LIN {X 0,Y 530.986,Z 634.341,A -85,B 0,C 180,E1 -4457.833,E2 -4457.833} C_VEL
LIN {X 0,Y 531.019,Z 634.341,A -85,B 0,C 180,E1 -4460.559,E2 -4460.559} C_VEL
LIN {X 0,Y 530.968,Z 634.345,A -85,B 0,C 180,E1 -4463.842,E2 -4463.842} C_VEL
LIN {X 0,Y 530.995,Z 634.341,A -85,B 0,C 180,E1 -4466.494,E2 -4466.494} C_VEL
LIN {X 0,Y 530.979,Z 634.341,A -85,B 0,C 180,E1 -4469.353,E2 -4469.353} C_VEL
LIN {X 0,Y 531.014,Z 634.337,A -85,B 0,C 180,E1 -4472.404,E2 -4472.404} C_VEL
LIN {X 0,Y 531.004,Z 634.337,A -85,B 0,C 180,E1 -4474.942,E2 -4474.942} C_VEL
LIN {X 0,Y 530.967,Z 634.342,A -85,B 0,C 180,E1 -4478.246,E2 -4478.246} C_VEL
LIN {X 0,Y 530.993,Z 634.339,A -85,B 0,C 180,E1 -4480.677,E2 -4480.677} C_VEL
LIN {X 0,Y 530.982,Z 634.346,A -85,B 0,C 180,E1 -4483.071,E2 -4483.071} C_VEL
LIN {X 0,Y 531.014,Z 634.339,A -85,B 0,C 180,E1 -4485.436,E2 -4485.436} C_VEL
LIN {X 0,Y 531.042,Z 634.337,A -85,B 0,C 180,E1 -4488.55,E2 -4488.55} C_VEL
LIN {X 0,Y 531.056,Z 634.331,A -85,B 0,C 180,E1 -4491.629,E2 -4491.629} C_VEL
LIN {X 0,Y 531.118,Z 634.33,A -85,B 0,C 180,E1 -4494.685,E2 -4494.685} C_VEL
LIN {X 0,Y 531.134,Z 634.323,A -85,B 0,C 180,E1 -4497.725,E2 -4497.725} C_VEL
LIN {X 0,Y 531.149,Z 634.323,A -85,B 0,C 180,E1 -4500.758,E2 -4500.758} C_VEL
LIN {X 0,Y 531.105,Z 634.328,A -85,B 0,C 180,E1 -4503.034,E2 -4503.034} C_VEL
LIN {X 0,Y 531.06,Z 634.46,A -85,B 0,C 180,E1 -4504.649,E2 -4504.649} C_VEL
LIN {X 0,Y 531.55,Z 640.442,A -85,B 0,C 180,E1 -4506.072,E2 -4506.072} C_VEL
LIN {X 0,Y 531.68,Z 653.246,A -85,B 0,C 180,E1 -4509.127,E2 -4509.127} C_VEL
LIN {X 0,Y 531.676,Z 665.851,A -85,B 0,C 180,E1 -4512.21,E2 -4512.21} C_VEL
LIN {X 0,Y 531.52,Z 677.588,A -85,B 0,C 180,E1 -4515.154,E2 -4515.154} C_VEL
LIN {X 0,Y 531.397,Z 689.132,A -85,B 0,C 180,E1 -4518.067,E2 -4518.067} C_VEL
LIN {X 0,Y 531.209,Z 700.198,A -85,B 0,C 180,E1 -4520.929,E2 -4520.929} C_VEL
LIN {X 0,Y 531.024,Z 710.926,A -85,B 0,C 180,E1 -4523.717,E2 -4523.717} C_VEL
LIN {X 0,Y 530.877,Z 722.756,A -85,B 0,C 180,E1 -4526.751,E2 -4526.751} C_VEL
LIN {X 0,Y 530.807,Z 725.673,A -85,B 0,C 180,E1 -4527.491,E2 -4527.491} C_VEL
LIN {X 0,Y 532.339,Z 736.306,A -85,B 0,C 180,E1 -4527.756,E2 -4527.756} C_VEL
LIN {X 0,Y 532.152,Z 749.102,A -85,B 0,C 180,E1 -4528.152,E2 -4528.152} C_VEL
LIN {X 0,Y 531.867,Z 762.095,A -85,B 0,C 180,E1 -4528.728,E2 -4528.728} C_VEL
LIN {X 0,Y 531.627,Z 773.458,A -85,B 0,C 180,E1 -4529.392,E2 -4529.392} C_VEL
LIN {X 0,Y 531.387,Z 783.981,A -85,B 0,C 180,E1 -4530.171,E2 -4530.171} C_VEL
LIN {X 0,Y 531.104,Z 794.919,A -85,B 0,C 180,E1 -4531.18,E2 -4531.18} C_VEL
LIN {X 0,Y 530.918,Z 804.119,A -85,B 0,C 180,E1 -4532.24,E2 -4532.24} C_VEL
LIN {X 0,Y 530.742,Z 812.635,A -85,B 0,C 180,E1 -4533.465,E2 -4533.465} C_VEL
LIN {X 0,Y 530.587,Z 819.541,A -85,B 0,C 180,E1 -4534.72,E2 -4534.72} C_VEL
LIN {X 0,Y 530.57,Z 820.437,A -85,B 0,C 180,E1 -4534.911,E2 -4534.911} C_VEL
LIN {X 0,Y 529.876,Z 823.006,A -85,B 0,C 180,E1 -4535.484,E2 -4535.484} C_VEL
LIN {X 0,Y 526.94,Z 826.619,A -85,B 0,C 180,E1 -4536.435,E2 -4536.435} C_VEL
LIN {X 0,Y 524.46,Z 828.999,A -85,B 0,C 180,E1 -4537.22,E2 -4537.22} C_VEL
LIN {X 0,Y 523.384,Z 830.509,A -85,B 0,C 180,E1 -4537.836,E2 -4537.836} C_VEL
LIN {X 0,Y 523.29,Z 830.939,A -85,B 0,C 180,E1 -4538.047,E2 -4538.047} C_VEL
LIN {X 0,Y 523.257,Z 832.782,A -85,B 0,C 180,E1 -4539.144,E2 -4539.144} C_VEL
LIN {X 0,Y 523.237,Z 833.705,A -85,B 0,C 180,E1 -4540.145,E2 -4540.145} C_VEL
LIN {X 0,Y 523.242,Z 833.97,A -85,B 0,C 180,E1 -4541.222,E2 -4541.222} C_VEL
LIN {X 0,Y 523.262,Z 833.392,A -85,B 0,C 180,E1 -4542.379,E2 -4542.379} C_VEL
LIN {X 0,Y 523.26,Z 831.963,A -85,B 0,C 180,E1 -4543.509,E2 -4543.509} C_VEL
LIN {X 0,Y 523.362,Z 828.741,A -85,B 0,C 180,E1 -4544.974,E2 -4544.974} C_VEL
LIN {X 0,Y 523.418,Z 825.122,A -85,B 0,C 180,E1 -4546.12,E2 -4546.12} C_VEL
LIN {X 0,Y 523.493,Z 820.639,A -85,B 0,C 180,E1 -4547.218,E2 -4547.218} C_VEL
LIN {X 0,Y 523.636,Z 813.716,A -85,B 0,C 180,E1 -4548.551,E2 -4548.551} C_VEL
LIN {X 0,Y 523.816,Z 806.45,A -85,B 0,C 180,E1 -4549.658,E2 -4549.658} C_VEL
LIN {X 0,Y 524.007,Z 797.164,A -85,B 0,C 180,E1 -4550.8,E2 -4550.8} C_VEL
LIN {X 0,Y 524.268,Z 787.013,A -85,B 0,C 180,E1 -4551.807,E2 -4551.807} C_VEL
LIN {X 0,Y 524.587,Z 775.831,A -85,B 0,C 180,E1 -4552.69,E2 -4552.69} C_VEL
LIN {X 0,Y 524.854,Z 764.914,A -85,B 0,C 180,E1 -4553.376,E2 -4553.376} C_VEL
LIN {X 0,Y 525.154,Z 753.694,A -85,B 0,C 180,E1 -4553.926,E2 -4553.926} C_VEL
LIN {X 0,Y 525.392,Z 740.78,A -85,B 0,C 180,E1 -4554.388,E2 -4554.388} C_VEL
LIN {X 0,Y 525.236,Z 734.832,A -85,B 0,C 180,E1 -4554.553,E2 -4554.553} C_VEL
LIN {X 0,Y 523.71,Z 725.662,A -85,B 0,C 180,E1 -4554.789,E2 -4554.789} C_VEL
LIN {X 0,Y 523.937,Z 714.498,A -85,B 0,C 180,E1 -4557.679,E2 -4557.679} C_VEL
LIN {X 0,Y 524.166,Z 703.144,A -85,B 0,C 180,E1 -4560.635,E2 -4560.635} C_VEL
LIN {X 0,Y 524.387,Z 690.741,A -85,B 0,C 180,E1 -4563.891,E2 -4563.891} C_VEL
LIN {X 0,Y 524.587,Z 679.935,A -85,B 0,C 180,E1 -4566.721,E2 -4566.721} C_VEL
LIN {X 0,Y 524.755,Z 668.733,A -85,B 0,C 180,E1 -4569.637,E2 -4569.637} C_VEL
LIN {X 0,Y 524.836,Z 657.835,A -85,B 0,C 180,E1 -4572.465,E2 -4572.465} C_VEL
LIN {X 0,Y 524.902,Z 647.071,A -85,B 0,C 180,E1 -4575.263,E2 -4575.263} C_VEL
LIN {X 0,Y 524.69,Z 639.508,A -85,B 0,C 180,E1 -4577.232,E2 -4577.232} C_VEL
LIN {X 0,Y 524.013,Z 635.215,A -85,B 0,C 180,E1 -4578.395,E2 -4578.395} C_VEL
LIN {X 0,Y 524.007,Z 635.217,A -85,B 0,C 180,E1 -4581.517,E2 -4581.517} C_VEL
LIN {X 0,Y 524.086,Z 635.205,A -85,B 0,C 180,E1 -4584.614,E2 -4584.614} C_VEL
LIN {X 0,Y 524.114,Z 635.202,A -85,B 0,C 180,E1 -4587.695,E2 -4587.695} C_VEL
LIN {X 0,Y 524.127,Z 635.201,A -85,B 0,C 180,E1 -4590.769,E2 -4590.769} C_VEL
LIN {X 0,Y 524.075,Z 635.206,A -85,B 0,C 180,E1 -4593.075,E2 -4593.075} C_VEL
LIN {X 0,Y 524.039,Z 635.21,A -85,B 0,C 180,E1 -4596.159,E2 -4596.159} C_VEL
LIN {X 0,Y 524.008,Z 635.215,A -85,B 0,C 180,E1 -4598.484,E2 -4598.484} C_VEL
LIN {X 0,Y 524.027,Z 635.211,A -85,B 0,C 180,E1 -4601.752,E2 -4601.752} C_VEL
LIN {X 0,Y 523.995,Z 635.216,A -85,B 0,C 180,E1 -4605.053,E2 -4605.053} C_VEL
LIN {X 0,Y 523.966,Z 635.222,A -85,B 0,C 180,E1 -4607.969,E2 -4607.969} C_VEL
LIN {X 0,Y 523.974,Z 635.22,A -85,B 0,C 180,E1 -4610.41,E2 -4610.41} C_VEL
LIN {X 0,Y 523.913,Z 635.226,A -85,B 0,C 180,E1 -4612.894,E2 -4612.894} C_VEL
LIN {X 0,Y 523.986,Z 635.218,A -85,B 0,C 180,E1 -4615.046,E2 -4615.046} C_VEL
LIN {X 0,Y 525.285,Z 640.908,A -85,B 0,C 180,E1 -4615.35,E2 -4615.35} C_VEL
LIN {X 0,Y 525.101,Z 651.029,A -85,B 0,C 180,E1 -4615.891,E2 -4615.891} C_VEL
LIN {X 0,Y 524.873,Z 660.697,A -85,B 0,C 180,E1 -4616.533,E2 -4616.533} C_VEL
LIN {X 0,Y 524.633,Z 670.141,A -85,B 0,C 180,E1 -4617.301,E2 -4617.301} C_VEL
LIN {X 0,Y 524.395,Z 679.151,A -85,B 0,C 180,E1 -4618.192,E2 -4618.192} C_VEL
LIN {X 0,Y 524.111,Z 688.658,A -85,B 0,C 180,E1 -4619.354,E2 -4619.354} C_VEL
LIN {X 0,Y 523.919,Z 695.663,A -85,B 0,C 180,E1 -4620.424,E2 -4620.424} C_VEL
LIN {X 0,Y 523.785,Z 701.653,A -85,B 0,C 180,E1 -4621.553,E2 -4621.553} C_VEL
LIN {X 0,Y 523.673,Z 705.684,A -85,B 0,C 180,E1 -4622.468,E2 -4622.468} C_VEL
LIN {X 0,Y 523.569,Z 709.83,A -85,B 0,C 180,E1 -4623.67,E2 -4623.67} C_VEL
LIN {X 0,Y 523.483,Z 713.171,A -85,B 0,C 180,E1 -4625.02,E2 -4625.02} C_VEL
LIN {X 0,Y 523.427,Z 715.227,A -85,B 0,C 180,E1 -4626.33,E2 -4626.33} C_VEL
LIN {X 0,Y 523.387,Z 716.143,A -85,B 0,C 180,E1 -4627.604,E2 -4627.604} C_VEL
LIN {X 0,Y 523.404,Z 716.016,A -85,B 0,C 180,E1 -4628.85,E2 -4628.85} C_VEL
LIN {X 0,Y 523.449,Z 714.846,A -85,B 0,C 180,E1 -4630.126,E2 -4630.126} C_VEL
LIN {X 0,Y 523.558,Z 711.98,A -85,B 0,C 180,E1 -4631.665,E2 -4631.665} C_VEL
LIN {X 0,Y 523.622,Z 708.87,A -85,B 0,C 180,E1 -4632.769,E2 -4632.769} C_VEL
LIN {X 0,Y 523.694,Z 704.835,A -85,B 0,C 180,E1 -4633.867,E2 -4633.867} C_VEL
LIN {X 0,Y 523.806,Z 699.797,A -85,B 0,C 180,E1 -4634.956,E2 -4634.956} C_VEL
LIN {X 0,Y 524.014,Z 692.971,A -85,B 0,C 180,E1 -4636.131,E2 -4636.131} C_VEL
LIN {X 0,Y 524.232,Z 685.14,A -85,B 0,C 180,E1 -4637.222,E2 -4637.222} C_VEL
LIN {X 0,Y 524.462,Z 677.321,A -85,B 0,C 180,E1 -4638.12,E2 -4638.12} C_VEL
LIN {X 0,Y 524.734,Z 668.237,A -85,B 0,C 180,E1 -4638.983,E2 -4638.983} C_VEL
LIN {X 0,Y 524.967,Z 658.567,A -85,B 0,C 180,E1 -4639.737,E2 -4639.737} C_VEL
LIN {X 0,Y 525.255,Z 646.597,A -85,B 0,C 180,E1 -4640.477,E2 -4640.477} C_VEL
LIN {X 0,Y 525.315,Z 640.243,A -85,B 0,C 180,E1 -4640.792,E2 -4640.792} C_VEL
LIN {X 0,Y 523.963,Z 635.219,A -85,B 0,C 180,E1 -4641.074,E2 -4641.074} C_VEL
LIN {X 0,Y 523.901,Z 635.227,A -85,B 0,C 180,E1 -4643.825,E2 -4643.825} C_VEL
LIN {X 0,Y 523.942,Z 635.217,A -85,B 0,C 180,E1 -4646.636,E2 -4646.636} C_VEL
LIN {X 0,Y 523.956,Z 635.22,A -85,B 0,C 180,E1 -4649.356,E2 -4649.356} C_VEL
LIN {X 0,Y 523.979,Z 635.213,A -85,B 0,C 180,E1 -4652.281,E2 -4652.281} C_VEL
LIN {X 0,Y 523.948,Z 635.215,A -85,B 0,C 180,E1 -4654.581,E2 -4654.581} C_VEL
LIN {X 0,Y 523.92,Z 635.224,A -85,B 0,C 180,E1 -4657.757,E2 -4657.757} C_VEL
LIN {X 0,Y 523.976,Z 635.213,A -85,B 0,C 180,E1 -4660.408,E2 -4660.408} C_VEL
LIN {X 0,Y 523.968,Z 635.212,A -85,B 0,C 180,E1 -4662.837,E2 -4662.837} C_VEL
LIN {X 0,Y 523.978,Z 635.213,A -85,B 0,C 180,E1 -4665.236,E2 -4665.236} C_VEL
LIN {X 0,Y 524.013,Z 635.208,A -85,B 0,C 180,E1 -4668.394,E2 -4668.394} C_VEL
LIN {X 0,Y 524.006,Z 635.21,A -85,B 0,C 180,E1 -4671.516,E2 -4671.516} C_VEL
LIN {X 0,Y 524.084,Z 635.199,A -85,B 0,C 180,E1 -4674.614,E2 -4674.614} C_VEL
LIN {X 0,Y 524.115,Z 635.195,A -85,B 0,C 180,E1 -4677.695,E2 -4677.695} C_VEL
LIN {X 0,Y 524.125,Z 635.19,A -85,B 0,C 180,E1 -4680.768,E2 -4680.768} C_VEL
LIN {X 0,Y 524.075,Z 635.198,A -85,B 0,C 180,E1 -4683.075,E2 -4683.075} C_VEL
LIN {X 0,Y 524.047,Z 635.209,A -85,B 0,C 180,E1 -4686.159,E2 -4686.159} C_VEL
LIN {X 0,Y 524.001,Z 635.205,A -85,B 0,C 180,E1 -4689.262,E2 -4689.262} C_VEL
LIN {X 0,Y 524.004,Z 635.21,A -85,B 0,C 180,E1 -4691.74,E2 -4691.74} C_VEL
LIN {X 0,Y 523.994,Z 635.209,A -85,B 0,C 180,E1 -4695.052,E2 -4695.052} C_VEL
LIN {X 0,Y 523.965,Z 635.216,A -85,B 0,C 180,E1 -4697.969,E2 -4697.969} C_VEL
LIN {X 0,Y 523.973,Z 635.219,A -85,B 0,C 180,E1 -4700.41,E2 -4700.41} C_VEL
LIN {X 0,Y 523.913,Z 635.221,A -85,B 0,C 180,E1 -4702.894,E2 -4702.894} C_VEL
LIN {X 0,Y 523.955,Z 635.213,A -85,B 0,C 180,E1 -4705.419,E2 -4705.419} C_VEL
LIN {X 0,Y 523.971,Z 635.215,A -85,B 0,C 180,E1 -4707.999,E2 -4707.999} C_VEL
LIN {X 0,Y 523.946,Z 635.22,A -85,B 0,C 180,E1 -4710.855,E2 -4710.855} C_VEL
LIN {X 0,Y 523.961,Z 635.214,A -85,B 0,C 180,E1 -4713.735,E2 -4713.735} C_VEL
LIN {X 0,Y 523.905,Z 635.228,A -85,B 0,C 180,E1 -4716.401,E2 -4716.401} C_VEL
LIN {X 0,Y 523.925,Z 635.222,A -85,B 0,C 180,E1 -4719.085,E2 -4719.085} C_VEL
LIN {X 0,Y 523.959,Z 635.217,A -85,B 0,C 180,E1 -4722.119,E2 -4722.119} C_VEL
LIN {X 0,Y 523.955,Z 635.218,A -85,B 0,C 180,E1 -4725.309,E2 -4725.309} C_VEL
LIN {X 0,Y 523.958,Z 635.225,A -85,B 0,C 180,E1 -4728.69,E2 -4728.69} C_VEL
LIN {X 0,Y 523.935,Z 635.298,A -85,B 0,C 180,E1 -4731.655,E2 -4731.655} C_VEL
LIN {X 0,Y 525.505,Z 643.564,A -85,B 0,C 180,E1 -4733.678,E2 -4733.678} C_VEL
LIN {X 0,Y 525.513,Z 652.078,A -85,B 0,C 180,E1 -4735.595,E2 -4735.595} C_VEL
LIN {X 0,Y 525.326,Z 665.745,A -85,B 0,C 180,E1 -4738.55,E2 -4738.55} C_VEL
LIN {X 0,Y 525.103,Z 680.614,A -85,B 0,C 180,E1 -4741.632,E2 -4741.632} C_VEL
LIN {X 0,Y 524.896,Z 695.386,A -85,B 0,C 180,E1 -4744.63,E2 -4744.63} C_VEL
LIN {X 0,Y 524.67,Z 709.448,A -85,B 0,C 180,E1 -4747.392,E2 -4747.392} C_VEL
LIN {X 0,Y 524.502,Z 723.369,A -85,B 0,C 180,E1 -4750.066,E2 -4750.066} C_VEL
LIN {X 0,Y 524.304,Z 735.606,A -85,B 0,C 180,E1 -4752.479,E2 -4752.479} C_VEL
LIN {X 0,Y 524.002,Z 751.098,A -85,B 0,C 180,E1 -4755.633,E2 -4755.633} C_VEL
LIN {X 0,Y 523.898,Z 754.155,A -85,B 0,C 180,E1 -4756.249,E2 -4756.249} C_VEL
LIN {X 0,Y 525.459,Z 765.504,A -85,B 0,C 180,E1 -4756.513,E2 -4756.513} C_VEL
LIN {X 0,Y 525.239,Z 778.157,A -85,B 0,C 180,E1 -4756.901,E2 -4756.901} C_VEL
LIN {X 0,Y 524.976,Z 790.481,A -85,B 0,C 180,E1 -4757.435,E2 -4757.435} C_VEL
LIN {X 0,Y 524.767,Z 802.28,A -85,B 0,C 180,E1 -4758.114,E2 -4758.114} C_VEL
LIN {X 0,Y 524.493,Z 812.916,A -85,B 0,C 180,E1 -4758.894,E2 -4758.894} C_VEL
LIN {X 0,Y 524.17,Z 822.595,A -85,B 0,C 180,E1 -4759.767,E2 -4759.767} C_VEL
LIN {X 0,Y 523.93,Z 831.41,A -85,B 0,C 180,E1 -4760.737,E2 -4760.737} C_VEL
LIN {X 0,Y 523.724,Z 840.001,A -85,B 0,C 180,E1 -4761.9,E2 -4761.9} C_VEL
LIN {X 0,Y 523.575,Z 846.867,A -85,B 0,C 180,E1 -4763.061,E2 -4763.061} C_VEL
LIN {X 0,Y 523.544,Z 852.363,A -85,B 0,C 180,E1 -4764.221,E2 -4764.221} C_VEL
LIN {X 0,Y 523.361,Z 856.676,A -85,B 0,C 180,E1 -4765.378,E2 -4765.378} C_VEL
LIN {X 0,Y 523.444,Z 858.96,A -85,B 0,C 180,E1 -4766.15,E2 -4766.15} C_VEL
LIN {X 0,Y 523.368,Z 860.809,A -85,B 0,C 180,E1 -4766.921,E2 -4766.921} C_VEL
LIN {X 0,Y 523.334,Z 862.196,A -85,B 0,C 180,E1 -4767.691,E2 -4767.691} C_VEL
LIN {X 0,Y 523.25,Z 863.786,A -85,B 0,C 180,E1 -4769.23,E2 -4769.23} C_VEL
LIN {X 0,Y 523.246,Z 864,A -85,B 0,C 180,E1 -4770,E2 -4770} C_VEL
LIN {X 0,Y 523.274,Z 863.184,A -85,B 0,C 180,E1 -4771.539,E2 -4771.539} C_VEL
LIN {X 0,Y 523.334,Z 862.195,A -85,B 0,C 180,E1 -4772.309,E2 -4772.309} C_VEL
LIN {X 0,Y 523.368,Z 860.808,A -85,B 0,C 180,E1 -4773.079,E2 -4773.079} C_VEL
LIN {X 0,Y 523.442,Z 857.896,A -85,B 0,C 180,E1 -4774.234,E2 -4774.234} C_VEL
LIN {X 0,Y 523.464,Z 853.951,A -85,B 0,C 180,E1 -4775.392,E2 -4775.392} C_VEL
LIN {X 0,Y 523.523,Z 848.729,A -85,B 0,C 180,E1 -4776.58,E2 -4776.58} C_VEL
LIN {X 0,Y 523.664,Z 842.469,A -85,B 0,C 180,E1 -4777.712,E2 -4777.712} C_VEL
LIN {X 0,Y 523.857,Z 834.481,A -85,B 0,C 180,E1 -4778.875,E2 -4778.875} C_VEL
LIN {X 0,Y 524.084,Z 826.338,A -85,B 0,C 180,E1 -4779.844,E2 -4779.844} C_VEL
LIN {X 0,Y 524.369,Z 816.404,A -85,B 0,C 180,E1 -4780.815,E2 -4780.815} C_VEL
LIN {X 0,Y 524.706,Z 805.138,A -85,B 0,C 180,E1 -4781.691,E2 -4781.691} C_VEL
LIN {X 0,Y 524.898,Z 794.181,A -85,B 0,C 180,E1 -4782.37,E2 -4782.37} C_VEL
LIN {X 0,Y 525.166,Z 781.994,A -85,B 0,C 180,E1 -4782.953,E2 -4782.953} C_VEL
LIN {X 0,Y 525.381,Z 769.202,A -85,B 0,C 180,E1 -4783.39,E2 -4783.39} C_VEL
LIN {X 0,Y 525.253,Z 762.824,A -85,B 0,C 180,E1 -4783.553,E2 -4783.553} C_VEL
LIN {X 0,Y 523.893,Z 754.037,A -85,B 0,C 180,E1 -4783.775,E2 -4783.775} C_VEL
LIN {X 0,Y 524.179,Z 739.364,A -85,B 0,C 180,E1 -4786.753,E2 -4786.753} C_VEL
LIN {X 0,Y 524.397,Z 727.385,A -85,B 0,C 180,E1 -4789.168,E2 -4789.168} C_VEL
LIN {X 0,Y 524.654,Z 712.688,A -85,B 0,C 180,E1 -4792.028,E2 -4792.028} C_VEL
LIN {X 0,Y 524.912,Z 698.108,A -85,B 0,C 180,E1 -4794.944,E2 -4794.944} C_VEL
LIN {X 0,Y 525.2,Z 683.359,A -85,B 0,C 180,E1 -4797.971,E2 -4797.971} C_VEL
LIN {X 0,Y 525.447,Z 668.438,A -85,B 0,C 180,E1 -4801.127,E2 -4801.127} C_VEL
LIN {X 0,Y 525.721,Z 656.968,A -85,B 0,C 180,E1 -4803.636,E2 -4803.636} C_VEL
LIN {X 0,Y 525.993,Z 646.437,A -85,B 0,C 180,E1 -4806.007,E2 -4806.007} C_VEL
LIN {X 0,Y 524.727,Z 639.152,A -85,B 0,C 180,E1 -4807.793,E2 -4807.793} C_VEL
LIN {X 0,Y 523.93,Z 635.225,A -85,B 0,C 180,E1 -4808.82,E2 -4808.82} C_VEL
LIN {X 0,Y 523.957,Z 635.219,A -85,B 0,C 180,E1 -4811.31,E2 -4811.31} C_VEL
LIN {X 0,Y 523.954,Z 635.223,A -85,B 0,C 180,E1 -4814.691,E2 -4814.691} C_VEL
LIN {X 0,Y 523.955,Z 635.217,A -85,B 0,C 180,E1 -4817.881,E2 -4817.881} C_VEL
LIN {X 0,Y 523.964,Z 635.216,A -85,B 0,C 180,E1 -4820.919,E2 -4820.919} C_VEL
LIN {X 0,Y 523.923,Z 635.222,A -85,B 0,C 180,E1 -4823.827,E2 -4823.827} C_VEL
LIN {X 0,Y 523.938,Z 635.219,A -85,B 0,C 180,E1 -4826.635,E2 -4826.635} C_VEL
LIN {X 0,Y 523.96,Z 635.215,A -85,B 0,C 180,E1 -4829.356,E2 -4829.356} C_VEL
LIN {X 0,Y 523.976,Z 635.215,A -85,B 0,C 180,E1 -4832.28,E2 -4832.28} C_VEL
LIN {X 0,Y 523.951,Z 635.214,A -85,B 0,C 180,E1 -4834.581,E2 -4834.581} C_VEL
LIN {X 0,Y 523.912,Z 635.224,A -85,B 0,C 180,E1 -4837.106,E2 -4837.106} C_VEL
LIN {X 0,Y 523.974,Z 635.214,A -85,B 0,C 180,E1 -4839.865,E2 -4839.865} C_VEL
LIN {X 0,Y 523.962,Z 635.217,A -85,B 0,C 180,E1 -4842.837,E2 -4842.837} C_VEL
LIN {X 0,Y 523.972,Z 635.219,A -85,B 0,C 180,E1 -4845.235,E2 -4845.235} C_VEL
LIN {X 0,Y 524.007,Z 635.211,A -85,B 0,C 180,E1 -4848.394,E2 -4848.394} C_VEL
LIN {X 0,Y 524.003,Z 635.21,A -85,B 0,C 180,E1 -4851.516,E2 -4851.516} C_VEL
LIN {X 0,Y 524.079,Z 635.207,A -85,B 0,C 180,E1 -4854.614,E2 -4854.614} C_VEL
LIN {X 0,Y 524.106,Z 635.198,A -85,B 0,C 180,E1 -4857.694,E2 -4857.694} C_VEL
LIN {X 0,Y 524.119,Z 635.199,A -85,B 0,C 180,E1 -4860.768,E2 -4860.768} C_VEL
LIN {X 0,Y 524.071,Z 635.204,A -85,B 0,C 180,E1 -4863.075,E2 -4863.075} C_VEL
LIN {X 0,Y 523.993,Z 635.307,A -85,B 0,C 180,E1 -4864.519,E2 -4864.519} C_VEL
LIN {X 0,Y 524.561,Z 640.51,A -85,B 0,C 180,E1 -4865.767,E2 -4865.767} C_VEL
LIN {X 0,Y 524.679,Z 653.419,A -85,B 0,C 180,E1 -4868.861,E2 -4868.861} C_VEL
LIN {X 0,Y 524.677,Z 666.566,A -85,B 0,C 180,E1 -4872.092,E2 -4872.092} C_VEL
LIN {X 0,Y 524.511,Z 679.181,A -85,B 0,C 180,E1 -4875.264,E2 -4875.264} C_VEL
LIN {X 0,Y 524.377,Z 691.326,A -85,B 0,C 180,E1 -4878.358,E2 -4878.358} C_VEL
LIN {X 0,Y 524.145,Z 702.328,A -85,B 0,C 180,E1 -4881.225,E2 -4881.225} C_VEL
LIN {X 0,Y 523.935,Z 713.688,A -85,B 0,C 180,E1 -4884.199,E2 -4884.199} C_VEL
LIN {X 0,Y 523.764,Z 725.522,A -85,B 0,C 180,E1 -4887.267,E2 -4887.267} C_VEL
LIN {X 0,Y 523.758,Z 725.704,A -85,B 0,C 180,E1 -4887.313,E2 -4887.313} C_VEL
LIN {X 0,Y 525.431,Z 736.746,A -85,B 0,C 180,E1 -4887.589,E2 -4887.589} C_VEL
LIN {X 0,Y 525.244,Z 749.173,A -85,B 0,C 180,E1 -4887.982,E2 -4887.982} C_VEL
LIN {X 0,Y 524.907,Z 762.357,A -85,B 0,C 180,E1 -4888.576,E2 -4888.576} C_VEL
LIN {X 0,Y 524.636,Z 774.364,A -85,B 0,C 180,E1 -4889.297,E2 -4889.297} C_VEL
LIN {X 0,Y 524.357,Z 785.722,A -85,B 0,C 180,E1 -4890.173,E2 -4890.173} C_VEL
LIN {X 0,Y 524.049,Z 796.18,A -85,B 0,C 180,E1 -4891.18,E2 -4891.18} C_VEL
LIN {X 0,Y 523.826,Z 805.481,A -85,B 0,C 180,E1 -4892.303,E2 -4892.303} C_VEL
LIN {X 0,Y 523.692,Z 812.755,A -85,B 0,C 180,E1 -4893.382,E2 -4893.382} C_VEL
LIN {X 0,Y 523.512,Z 819.711,A -85,B 0,C 180,E1 -4894.67,E2 -4894.67} C_VEL
LIN {X 0,Y 523.427,Z 824.275,A -85,B 0,C 180,E1 -4895.737,E2 -4895.737} C_VEL
LIN {X 0,Y 523.363,Z 828.905,A -85,B 0,C 180,E1 -4897.177,E2 -4897.177} C_VEL
LIN {X 0,Y 523.29,Z 830.939,A -85,B 0,C 180,E1 -4898.047,E2 -4898.047} C_VEL
LIN {X 0,Y 522.591,Z 832.135,A -85,B 0,C 180,E1 -4898.676,E2 -4898.676} C_VEL
LIN {X 0,Y 519.675,Z 833.399,A -85,B 0,C 180,E1 -4899.709,E2 -4899.709} C_VEL
LIN {X 0,Y 517.234,Z 833.906,A -85,B 0,C 180,E1 -4900.548,E2 -4900.548} C_VEL
LIN {X 0,Y 516.204,Z 833.976,A -85,B 0,C 180,E1 -4901.198,E2 -4901.198} C_VEL
LIN {X 0,Y 516.13,Z 833.919,A -85,B 0,C 180,E1 -4901.417,E2 -4901.417} C_VEL
LIN {X 0,Y 516.167,Z 832.873,A -85,B 0,C 180,E1 -4902.905,E2 -4902.905} C_VEL
LIN {X 0,Y 516.259,Z 830.16,A -85,B 0,C 180,E1 -4904.454,E2 -4904.454} C_VEL
LIN {X 0,Y 516.287,Z 827.242,A -85,B 0,C 180,E1 -4905.55,E2 -4905.55} C_VEL
LIN {X 0,Y 516.367,Z 823.42,A -85,B 0,C 180,E1 -4906.645,E2 -4906.645} C_VEL
LIN {X 0,Y 516.458,Z 817.48,A -85,B 0,C 180,E1 -4907.962,E2 -4907.962} C_VEL
LIN {X 0,Y 516.637,Z 810.147,A -85,B 0,C 180,E1 -4909.236,E2 -4909.236} C_VEL
LIN {X 0,Y 516.893,Z 801.494,A -85,B 0,C 180,E1 -4910.424,E2 -4910.424} C_VEL
LIN {X 0,Y 517.164,Z 791.855,A -85,B 0,C 180,E1 -4911.496,E2 -4911.496} C_VEL
LIN {X 0,Y 517.505,Z 781.147,A -85,B 0,C 180,E1 -4912.447,E2 -4912.447} C_VEL
LIN {X 0,Y 517.768,Z 770.459,A -85,B 0,C 180,E1 -4913.211,E2 -4913.211} C_VEL
LIN {X 0,Y 518.108,Z 759.334,A -85,B 0,C 180,E1 -4913.839,E2 -4913.839} C_VEL
LIN {X 0,Y 518.371,Z 746.366,A -85,B 0,C 180,E1 -4914.387,E2 -4914.387} C_VEL
LIN {X 0,Y 518.377,Z 735.954,A -85,B 0,C 180,E1 -4914.707,E2 -4914.707} C_VEL
LIN {X 0,Y 516.678,Z 725.63,A -85,B 0,C 180,E1 -4914.988,E2 -4914.988} C_VEL
LIN {X 0,Y 516.888,Z 714.317,A -85,B 0,C 180,E1 -4917.977,E2 -4917.977} C_VEL
LIN {X 0,Y 517.162,Z 702.217,A -85,B 0,C 180,E1 -4921.157,E2 -4921.157} C_VEL
LIN {X 0,Y 517.385,Z 690.564,A -85,B 0,C 180,E1 -4924.236,E2 -4924.236} C_VEL
LIN {X 0,Y 517.586,Z 678.462,A -85,B 0,C 180,E1 -4927.418,E2 -4927.418} C_VEL
LIN {X 0,Y 517.756,Z 667.993,A -85,B 0,C 180,E1 -4930.163,E2 -4930.163} C_VEL
LIN {X 0,Y 517.858,Z 657.044,A -85,B 0,C 180,E1 -4933.036,E2 -4933.036} C_VEL
LIN {X 0,Y 517.933,Z 646.22,A -85,B 0,C 180,E1 -4935.863,E2 -4935.863} C_VEL
LIN {X 0,Y 517.66,Z 640.188,A -85,B 0,C 180,E1 -4937.455,E2 -4937.455} C_VEL
LIN {X 0,Y 516.968,Z 636.092,A -85,B 0,C 180,E1 -4938.582,E2 -4938.582} C_VEL
LIN {X 0,Y 516.972,Z 636.092,A -85,B 0,C 180,E1 -4941.4,E2 -4941.4} C_VEL
LIN {X 0,Y 517.012,Z 636.087,A -85,B 0,C 180,E1 -4943.757,E2 -4943.757} C_VEL
LIN {X 0,Y 517.086,Z 636.077,A -85,B 0,C 180,E1 -4947.664,E2 -4947.664} C_VEL
LIN {X 0,Y 517.097,Z 636.077,A -85,B 0,C 180,E1 -4950.779,E2 -4950.779} C_VEL
LIN {X 0,Y 517.016,Z 636.085,A -85,B 0,C 180,E1 -4953.117,E2 -4953.117} C_VEL
LIN {X 0,Y 517.004,Z 636.086,A -85,B 0,C 180,E1 -4956.244,E2 -4956.244} C_VEL
LIN {X 0,Y 516.956,Z 636.09,A -85,B 0,C 180,E1 -4959.39,E2 -4959.39} C_VEL
LIN {X 0,Y 516.986,Z 636.088,A -85,B 0,C 180,E1 -4961.824,E2 -4961.824} C_VEL
LIN {X 0,Y 516.947,Z 636.094,A -85,B 0,C 180,E1 -4965.147,E2 -4965.147} C_VEL
LIN {X 0,Y 516.927,Z 636.097,A -85,B 0,C 180,E1 -4968.222,E2 -4968.222} C_VEL
LIN {X 0,Y 516.914,Z 636.101,A -85,B 0,C 180,E1 -4970.702,E2 -4970.702} C_VEL
LIN {X 0,Y 516.897,Z 636.1,A -85,B 0,C 180,E1 -4974.073,E2 -4974.073} C_VEL
LIN {X 0,Y 516.939,Z 636.097,A -85,B 0,C 180,E1 -4974.866,E2 -4974.866} C_VEL
LIN {X 0,Y 518.381,Z 641.786,A -85,B 0,C 180,E1 -4975.174,E2 -4975.174} C_VEL
LIN {X 0,Y 518.182,Z 653.512,A -85,B 0,C 180,E1 -4975.82,E2 -4975.82} C_VEL
LIN {X 0,Y 517.879,Z 664.653,A -85,B 0,C 180,E1 -4976.605,E2 -4976.605} C_VEL
LIN {X 0,Y 517.606,Z 674.727,A -85,B 0,C 180,E1 -4977.494,E2 -4977.494} C_VEL
LIN {X 0,Y 517.356,Z 683.016,A -85,B 0,C 180,E1 -4978.389,E2 -4978.389} C_VEL
LIN {X 0,Y 517.087,Z 691.818,A -85,B 0,C 180,E1 -4979.558,E2 -4979.558} C_VEL
LIN {X 0,Y 516.898,Z 698.358,A -85,B 0,C 180,E1 -4980.628,E2 -4980.628} C_VEL
LIN {X 0,Y 516.735,Z 704.183,A -85,B 0,C 180,E1 -4981.805,E2 -4981.805} C_VEL
LIN {X 0,Y 516.627,Z 708.744,A -85,B 0,C 180,E1 -4982.966,E2 -4982.966} C_VEL
LIN {X 0,Y 516.527,Z 712.912,A -85,B 0,C 180,E1 -4984.379,E2 -4984.379} C_VEL
LIN {X 0,Y 516.43,Z 715.658,A -85,B 0,C 180,E1 -4985.816,E2 -4985.816} C_VEL
LIN {X 0,Y 516.406,Z 716.76,A -85,B 0,C 180,E1 -4986.785,E2 -4986.785} C_VEL
LIN {X 0,Y 516.376,Z 717.252,A -85,B 0,C 180,E1 -4987.871,E2 -4987.871} C_VEL
LIN {X 0,Y 516.421,Z 716.909,A -85,B 0,C 180,E1 -4989.13,E2 -4989.13} C_VEL
LIN {X 0,Y 516.466,Z 714.91,A -85,B 0,C 180,E1 -4990.782,E2 -4990.782} C_VEL
LIN {X 0,Y 516.557,Z 712.767,A -85,B 0,C 180,E1 -4991.811,E2 -4991.811} C_VEL
LIN {X 0,Y 516.634,Z 709.829,A -85,B 0,C 180,E1 -4992.857,E2 -4992.857} C_VEL
LIN {X 0,Y 516.74,Z 704.818,A -85,B 0,C 180,E1 -4994.19,E2 -4994.19} C_VEL
LIN {X 0,Y 516.885,Z 699.652,A -85,B 0,C 180,E1 -4995.27,E2 -4995.27} C_VEL
LIN {X 0,Y 517.072,Z 693.064,A -85,B 0,C 180,E1 -4996.387,E2 -4996.387} C_VEL
LIN {X 0,Y 517.326,Z 685.149,A -85,B 0,C 180,E1 -4997.479,E2 -4997.479} C_VEL
LIN {X 0,Y 517.585,Z 676.965,A -85,B 0,C 180,E1 -4998.405,E2 -4998.405} C_VEL
LIN {X 0,Y 517.912,Z 666.667,A -85,B 0,C 180,E1 -4999.356,E2 -4999.356} C_VEL
LIN {X 0,Y 518.18,Z 655.943,A -85,B 0,C 180,E1 -5000.145,E2 -5000.145} C_VEL
LIN {X 0,Y 518.393,Z 644.103,A -85,B 0,C 180,E1 -5000.827,E2 -5000.827} C_VEL
LIN {X 0,Y 518.171,Z 640.542,A -85,B 0,C 180,E1 -5001.009,E2 -5001.009} C_VEL
LIN {X 0,Y 516.913,Z 636.099,A -85,B 0,C 180,E1 -5001.254,E2 -5001.254} C_VEL
LIN {X 0,Y 516.872,Z 636.099,A -85,B 0,C 180,E1 -5004.22,E2 -5004.22} C_VEL
LIN {X 0,Y 516.895,Z 636.097,A -85,B 0,C 180,E1 -5007.053,E2 -5007.053} C_VEL
LIN {X 0,Y 516.893,Z 636.101,A -85,B 0,C 180,E1 -5009.796,E2 -5009.796} C_VEL
LIN {X 0,Y 516.929,Z 636.09,A -85,B 0,C 180,E1 -5012.467,E2 -5012.467} C_VEL
LIN {X 0,Y 516.876,Z 636.097,A -85,B 0,C 180,E1 -5015.07,E2 -5015.07} C_VEL
LIN {X 0,Y 516.869,Z 636.101,A -85,B 0,C 180,E1 -5017.622,E2 -5017.622} C_VEL
LIN {X 0,Y 516.933,Z 636.094,A -85,B 0,C 180,E1 -5020.13,E2 -5020.13} C_VEL
LIN {X 0,Y 516.93,Z 636.089,A -85,B 0,C 180,E1 -5022.596,E2 -5022.596} C_VEL
LIN {X 0,Y 516.943,Z 636.088,A -85,B 0,C 180,E1 -5025.03,E2 -5025.03} C_VEL
LIN {X 0,Y 516.967,Z 636.087,A -85,B 0,C 180,E1 -5028.234,E2 -5028.234} C_VEL
LIN {X 0,Y 516.971,Z 636.086,A -85,B 0,C 180,E1 -5031.4,E2 -5031.4} C_VEL
LIN {X 0,Y 517.011,Z 636.083,A -85,B 0,C 180,E1 -5033.757,E2 -5033.757} C_VEL
LIN {X 0,Y 517.087,Z 636.07,A -85,B 0,C 180,E1 -5037.663,E2 -5037.663} C_VEL
LIN {X 0,Y 517.095,Z 636.066,A -85,B 0,C 180,E1 -5040.779,E2 -5040.779} C_VEL
LIN {X 0,Y 517.016,Z 636.078,A -85,B 0,C 180,E1 -5043.117,E2 -5043.117} C_VEL
LIN {X 0,Y 517.011,Z 636.087,A -85,B 0,C 180,E1 -5046.243,E2 -5046.243} C_VEL
LIN {X 0,Y 516.955,Z 636.083,A -85,B 0,C 180,E1 -5049.389,E2 -5049.389} C_VEL
LIN {X 0,Y 516.954,Z 636.089,A -85,B 0,C 180,E1 -5051.807,E2 -5051.807} C_VEL
LIN {X 0,Y 516.946,Z 636.087,A -85,B 0,C 180,E1 -5055.147,E2 -5055.147} C_VEL
LIN {X 0,Y 516.926,Z 636.096,A -85,B 0,C 180,E1 -5058.222,E2 -5058.222} C_VEL
LIN {X 0,Y 516.914,Z 636.095,A -85,B 0,C 180,E1 -5060.702,E2 -5060.702} C_VEL
LIN {X 0,Y 516.905,Z 636.095,A -85,B 0,C 180,E1 -5064.072,E2 -5064.072} C_VEL
LIN {X 0,Y 516.928,Z 636.096,A -85,B 0,C 180,E1 -5066.658,E2 -5066.658} C_VEL
LIN {X 0,Y 516.913,Z 636.092,A -85,B 0,C 180,E1 -5069.524,E2 -5069.524} C_VEL
LIN {X 0,Y 516.897,Z 636.101,A -85,B 0,C 180,E1 -5072.543,E2 -5072.543} C_VEL
LIN {X 0,Y 516.868,Z 636.099,A -85,B 0,C 180,E1 -5075.33,E2 -5075.33} C_VEL
LIN {X 0,Y 516.883,Z 636.098,A -85,B 0,C 180,E1 -5077.943,E2 -5077.943} C_VEL
LIN {X 0,Y 516.898,Z 636.102,A -85,B 0,C 180,E1 -5080.741,E2 -5080.741} C_VEL
LIN {X 0,Y 516.885,Z 636.096,A -85,B 0,C 180,E1 -5083.893,E2 -5083.893} C_VEL
LIN {X 0,Y 516.884,Z 636.099,A -85,B 0,C 180,E1 -5086.107,E2 -5086.107} C_VEL
LIN {X 0,Y 516.916,Z 636.1,A -85,B 0,C 180,E1 -5088.399,E2 -5088.399} C_VEL
LIN {X 0,Y 516.922,Z 636.258,A -85,B 0,C 180,E1 -5091.432,E2 -5091.432} C_VEL
LIN {X 0,Y 518.585,Z 645.077,A -85,B 0,C 180,E1 -5093.636,E2 -5093.636} C_VEL
LIN {X 0,Y 518.61,Z 652.382,A -85,B 0,C 180,E1 -5095.308,E2 -5095.308} C_VEL
LIN {X 0,Y 518.334,Z 666.49,A -85,B 0,C 180,E1 -5098.418,E2 -5098.418} C_VEL
LIN {X 0,Y 518.101,Z 680.747,A -85,B 0,C 180,E1 -5101.434,E2 -5101.434} C_VEL
LIN {X 0,Y 517.863,Z 694.477,A -85,B 0,C 180,E1 -5104.26,E2 -5104.26} C_VEL
LIN {X 0,Y 517.676,Z 707.119,A -85,B 0,C 180,E1 -5106.814,E2 -5106.814} C_VEL
LIN {X 0,Y 517.432,Z 722.776,A -85,B 0,C 180,E1 -5109.865,E2 -5109.865} C_VEL
LIN {X 0,Y 517.187,Z 737.957,A -85,B 0,C 180,E1 -5112.809,E2 -5112.809} C_VEL
LIN {X 0,Y 516.967,Z 751.098,A -85,B 0,C 180,E1 -5115.433,E2 -5115.433} C_VEL
LIN {X 0,Y 516.883,Z 754.155,A -85,B 0,C 180,E1 -5116.059,E2 -5116.059} C_VEL
LIN {X 0,Y 518.579,Z 765.503,A -85,B 0,C 180,E1 -5116.33,E2 -5116.33} C_VEL
LIN {X 0,Y 518.317,Z 778.156,A -85,B 0,C 180,E1 -5116.723,E2 -5116.723} C_VEL
LIN {X 0,Y 518.043,Z 790.48,A -85,B 0,C 180,E1 -5117.264,E2 -5117.264} C_VEL
LIN {X 0,Y 517.809,Z 801.915,A -85,B 0,C 180,E1 -5117.928,E2 -5117.928} C_VEL
LIN {X 0,Y 517.521,Z 812.914,A -85,B 0,C 180,E1 -5118.742,E2 -5118.742} C_VEL
LIN {X 0,Y 517.17,Z 822.594,A -85,B 0,C 180,E1 -5119.626,E2 -5119.626} C_VEL
LIN {X 0,Y 516.9,Z 831.41,A -85,B 0,C 180,E1 -5120.609,E2 -5120.609} C_VEL
LIN {X 0,Y 516.683,Z 840.001,A -85,B 0,C 180,E1 -5121.788,E2 -5121.788} C_VEL
LIN {X 0,Y 516.507,Z 846.867,A -85,B 0,C 180,E1 -5122.965,E2 -5122.965} C_VEL
LIN {X 0,Y 516.454,Z 852.363,A -85,B 0,C 180,E1 -5124.142,E2 -5124.142} C_VEL
LIN {X 0,Y 516.272,Z 856.675,A -85,B 0,C 180,E1 -5125.315,E2 -5125.315} C_VEL
LIN {X 0,Y 516.355,Z 858.959,A -85,B 0,C 180,E1 -5126.097,E2 -5126.097} C_VEL
LIN {X 0,Y 516.283,Z 860.809,A -85,B 0,C 180,E1 -5126.878,E2 -5126.878} C_VEL
LIN {X 0,Y 516.26,Z 862.196,A -85,B 0,C 180,E1 -5127.659,E2 -5127.659} C_VEL
LIN {X 0,Y 516.16,Z 863.786,A -85,B 0,C 180,E1 -5129.219,E2 -5129.219} C_VEL
LIN {X 0,Y 516.154,Z 864,A -85,B 0,C 180,E1 -5130,E2 -5130} C_VEL
LIN {X 0,Y 516.191,Z 863.183,A -85,B 0,C 180,E1 -5131.56,E2 -5131.56} C_VEL
LIN {X 0,Y 516.26,Z 862.195,A -85,B 0,C 180,E1 -5132.34,E2 -5132.34} C_VEL
LIN {X 0,Y 516.282,Z 860.808,A -85,B 0,C 180,E1 -5133.121,E2 -5133.121} C_VEL
LIN {X 0,Y 516.344,Z 857.896,A -85,B 0,C 180,E1 -5134.293,E2 -5134.293} C_VEL
LIN {X 0,Y 516.405,Z 853.951,A -85,B 0,C 180,E1 -5135.466,E2 -5135.466} C_VEL
LIN {X 0,Y 516.486,Z 848.036,A -85,B 0,C 180,E1 -5136.807,E2 -5136.807} C_VEL
LIN {X 0,Y 516.64,Z 841.238,A -85,B 0,C 180,E1 -5138.015,E2 -5138.015} C_VEL
LIN {X 0,Y 516.867,Z 832.996,A -85,B 0,C 180,E1 -5139.193,E2 -5139.193} C_VEL
LIN {X 0,Y 517.079,Z 824.544,A -85,B 0,C 180,E1 -5140.177,E2 -5140.177} C_VEL
LIN {X 0,Y 517.447,Z 814.098,A -85,B 0,C 180,E1 -5141.159,E2 -5141.159} C_VEL
LIN {X 0,Y 517.744,Z 802.428,A -85,B 0,C 180,E1 -5142.039,E2 -5142.039} C_VEL
LIN {X 0,Y 518.043,Z 790.5,A -85,B 0,C 180,E1 -5142.735,E2 -5142.735} C_VEL
LIN {X 0,Y 518.31,Z 778.188,A -85,B 0,C 180,E1 -5143.277,E2 -5143.277} C_VEL
LIN {X 0,Y 518.56,Z 765.06,A -85,B 0,C 180,E1 -5143.682,E2 -5143.682} C_VEL
LIN {X 0,Y 516.878,Z 754.037,A -85,B 0,C 180,E1 -5143.966,E2 -5143.966} C_VEL
LIN {X 0,Y 517.132,Z 741.114,A -85,B 0,C 180,E1 -5146.582,E2 -5146.582} C_VEL
LIN {X 0,Y 517.387,Z 725.507,A -85,B 0,C 180,E1 -5149.645,E2 -5149.645} C_VEL
LIN {X 0,Y 517.586,Z 711.834,A -85,B 0,C 180,E1 -5152.345,E2 -5152.345} C_VEL
LIN {X 0,Y 517.914,Z 697.405,A -85,B 0,C 180,E1 -5155.305,E2 -5155.305} C_VEL
LIN {X 0,Y 518.197,Z 683.659,A -85,B 0,C 180,E1 -5158.169,E2 -5158.169} C_VEL
LIN {X 0,Y 518.491,Z 670.488,A -85,B 0,C 180,E1 -5161.002,E2 -5161.002} C_VEL
LIN {X 0,Y 518.853,Z 656.926,A -85,B 0,C 180,E1 -5164.01,E2 -5164.01} C_VEL
LIN {X 0,Y 519.093,Z 647.916,A -85,B 0,C 180,E1 -5166.081,E2 -5166.081} C_VEL
LIN {X 0,Y 518.028,Z 641.679,A -85,B 0,C 180,E1 -5167.625,E2 -5167.625} C_VEL
LIN {X 0,Y 516.886,Z 636.103,A -85,B 0,C 180,E1 -5169.1,E2 -5169.1} C_VEL
LIN {X 0,Y 516.911,Z 636.095,A -85,B 0,C 180,E1 -5171.774,E2 -5171.774} C_VEL
LIN {X 0,Y 516.92,Z 636.096,A -85,B 0,C 180,E1 -5175.009,E2 -5175.009} C_VEL
LIN {X 0,Y 516.92,Z 636.099,A -85,B 0,C 180,E1 -5178.397,E2 -5178.397} C_VEL
LIN {X 0,Y 516.906,Z 636.093,A -85,B 0,C 180,E1 -5181.286,E2 -5181.286} C_VEL
LIN {X 0,Y 516.885,Z 636.102,A -85,B 0,C 180,E1 -5184.221,E2 -5184.221} C_VEL
LIN {X 0,Y 516.892,Z 636.095,A -85,B 0,C 180,E1 -5187.053,E2 -5187.053} C_VEL
LIN {X 0,Y 516.898,Z 636.101,A -85,B 0,C 180,E1 -5189.796,E2 -5189.796} C_VEL
LIN {X 0,Y 516.926,Z 636.092,A -85,B 0,C 180,E1 -5192.467,E2 -5192.467} C_VEL
LIN {X 0,Y 516.907,Z 636.094,A -85,B 0,C 180,E1 -5195.072,E2 -5195.072} C_VEL
LIN {X 0,Y 516.882,Z 636.097,A -85,B 0,C 180,E1 -5198.462,E2 -5198.462} C_VEL
LIN {X 0,Y 516.9,Z 636.097,A -85,B 0,C 180,E1 -5200.955,E2 -5200.955} C_VEL
LIN {X 0,Y 516.909,Z 636.098,A -85,B 0,C 180,E1 -5203.41,E2 -5203.41} C_VEL
LIN {X 0,Y 516.891,Z 636.096,A -85,B 0,C 180,E1 -5205.833,E2 -5205.833} C_VEL
LIN {X 0,Y 516.999,Z 636.083,A -85,B 0,C 180,E1 -5208.234,E2 -5208.234} C_VEL
LIN {X 0,Y 516.968,Z 636.087,A -85,B 0,C 180,E1 -5211.4,E2 -5211.4} C_VEL
LIN {X 0,Y 517.004,Z 636.083,A -85,B 0,C 180,E1 -5213.757,E2 -5213.757} C_VEL
LIN {X 0,Y 517.078,Z 636.074,A -85,B 0,C 180,E1 -5217.663,E2 -5217.663} C_VEL
LIN {X 0,Y 517.089,Z 636.075,A -85,B 0,C 180,E1 -5220.779,E2 -5220.779} C_VEL
LIN {X 0,Y 517.012,Z 636.084,A -85,B 0,C 180,E1 -5223.117,E2 -5223.117} C_VEL
LIN {X 0,Y 516.942,Z 636.177,A -85,B 0,C 180,E1 -5224.386,E2 -5224.386} C_VEL
LIN {X 0,Y 517.517,Z 640.589,A -85,B 0,C 180,E1 -5225.455,E2 -5225.455} C_VEL
LIN {X 0,Y 517.647,Z 651.969,A -85,B 0,C 180,E1 -5228.196,E2 -5228.196} C_VEL
LIN {X 0,Y 517.643,Z 663.21,A -85,B 0,C 180,E1 -5230.957,E2 -5230.957} C_VEL
LIN {X 0,Y 517.576,Z 672.755,A -85,B 0,C 180,E1 -5233.346,E2 -5233.346} C_VEL
LIN {X 0,Y 517.44,Z 683.808,A -85,B 0,C 180,E1 -5236.167,E2 -5236.167} C_VEL
LIN {X 0,Y 517.281,Z 694.994,A -85,B 0,C 180,E1 -5239.031,E2 -5239.031} C_VEL
LIN {X 0,Y 517.065,Z 706.035,A -85,B 0,C 180,E1 -5241.949,E2 -5241.949} C_VEL
LIN {X 0,Y 516.895,Z 716.188,A -85,B 0,C 180,E1 -5244.602,E2 -5244.602} C_VEL
LIN {X 0,Y 516.721,Z 725.64,A -85,B 0,C 180,E1 -5247.106,E2 -5247.106} C_VEL
LIN {X 0,Y 518.513,Z 738.093,A -85,B 0,C 180,E1 -5247.441,E2 -5247.441} C_VEL
LIN {X 0,Y 518.248,Z 751.417,A -85,B 0,C 180,E1 -5247.895,E2 -5247.895} C_VEL
LIN {X 0,Y 517.949,Z 763.46,A -85,B 0,C 180,E1 -5248.464,E2 -5248.464} C_VEL
LIN {X 0,Y 517.658,Z 774.515,A -85,B 0,C 180,E1 -5249.147,E2 -5249.147} C_VEL
LIN {X 0,Y 517.356,Z 785.712,A -85,B 0,C 180,E1 -5250.023,E2 -5250.023} C_VEL
LIN {X 0,Y 517.047,Z 795.971,A -85,B 0,C 180,E1 -5251.022,E2 -5251.022} C_VEL
LIN {X 0,Y 516.808,Z 804.35,A -85,B 0,C 180,E1 -5252.029,E2 -5252.029} C_VEL
LIN {X 0,Y 516.632,Z 812.272,A -85,B 0,C 180,E1 -5253.198,E2 -5253.198} C_VEL
LIN {X 0,Y 516.472,Z 818.756,A -85,B 0,C 180,E1 -5254.383,E2 -5254.383} C_VEL
LIN {X 0,Y 516.334,Z 824.847,A -85,B 0,C 180,E1 -5255.823,E2 -5255.823} C_VEL
LIN {X 0,Y 516.279,Z 829.333,A -85,B 0,C 180,E1 -5257.284,E2 -5257.284} C_VEL
LIN {X 0,Y 516.173,Z 832.303,A -85,B 0,C 180,E1 -5258.779,E2 -5258.779} C_VEL
LIN {X 0,Y 516.146,Z 833.815,A -85,B 0,C 180,E1 -5260.315,E2 -5260.315} C_VEL
LIN {X 0,Y 516.13,Z 833.919,A -85,B 0,C 180,E1 -5261.417,E2 -5261.417} C_VEL
LIN {X 0,Y 515.494,Z 833.724,A -85,B 0,C 180,E1 -5262.07,E2 -5262.07} C_VEL
LIN {X 0,Y 512.678,Z 832.752,A -85,B 0,C 180,E1 -5263.125,E2 -5263.125} C_VEL
LIN {X 0,Y 510.287,Z 831.371,A -85,B 0,C 180,E1 -5263.965,E2 -5263.965} C_VEL
LIN {X 0,Y 509.261,Z 829.964,A -85,B 0,C 180,E1 -5264.605,E2 -5264.605} C_VEL
LIN {X 0,Y 509.178,Z 829.422,A -85,B 0,C 180,E1 -5264.82,E2 -5264.82} C_VEL
LIN {X 0,Y 509.273,Z 824.735,A -85,B 0,C 180,E1 -5266.371,E2 -5266.371} C_VEL
LIN {X 0,Y 509.347,Z 820.323,A -85,B 0,C 180,E1 -5267.461,E2 -5267.461} C_VEL
LIN {X 0,Y 509.506,Z 813.763,A -85,B 0,C 180,E1 -5268.752,E2 -5268.752} C_VEL
LIN {X 0,Y 509.713,Z 806.802,A -85,B 0,C 180,E1 -5269.849,E2 -5269.849} C_VEL
LIN {X 0,Y 509.939,Z 798.547,A -85,B 0,C 180,E1 -5270.912,E2 -5270.912} C_VEL
LIN {X 0,Y 510.248,Z 788.415,A -85,B 0,C 180,E1 -5271.974,E2 -5271.974} C_VEL
LIN {X 0,Y 510.642,Z 777.606,A -85,B 0,C 180,E1 -5272.883,E2 -5272.883} C_VEL
LIN {X 0,Y 510.957,Z 765.567,A -85,B 0,C 180,E1 -5273.68,E2 -5273.68} C_VEL
LIN {X 0,Y 511.332,Z 753.919,A -85,B 0,C 180,E1 -5274.272,E2 -5274.272} C_VEL
LIN {X 0,Y 511.574,Z 741.426,A -85,B 0,C 180,E1 -5274.736,E2 -5274.736} C_VEL
LIN {X 0,Y 511.478,Z 736.801,A -85,B 0,C 180,E1 -5274.874,E2 -5274.874} C_VEL
LIN {X 0,Y 509.618,Z 725.714,A -85,B 0,C 180,E1 -5275.179,E2 -5275.179} C_VEL
LIN {X 0,Y 509.862,Z 715.376,A -85,B 0,C 180,E1 -5277.949,E2 -5277.949} C_VEL
LIN {X 0,Y 510.144,Z 703.22,A -85,B 0,C 180,E1 -5281.173,E2 -5281.173} C_VEL
LIN {X 0,Y 510.385,Z 691.46,A -85,B 0,C 180,E1 -5284.295,E2 -5284.295} C_VEL
LIN {X 0,Y 510.576,Z 679.993,A -85,B 0,C 180,E1 -5287.331,E2 -5287.331} C_VEL
LIN {X 0,Y 510.785,Z 668.759,A -85,B 0,C 180,E1 -5290.3,E2 -5290.3} C_VEL
LIN {X 0,Y 510.91,Z 659.331,A -85,B 0,C 180,E1 -5292.798,E2 -5292.798} C_VEL
LIN {X 0,Y 510.986,Z 648.438,A -85,B 0,C 180,E1 -5295.667,E2 -5295.667} C_VEL
LIN {X 0,Y 510.773,Z 642.349,A -85,B 0,C 180,E1 -5297.283,E2 -5297.283} C_VEL
LIN {X 0,Y 509.92,Z 636.968,A -85,B 0,C 180,E1 -5298.787,E2 -5298.787} C_VEL
LIN {X 0,Y 509.953,Z 636.964,A -85,B 0,C 180,E1 -5302.079,E2 -5302.079} C_VEL
LIN {X 0,Y 509.985,Z 636.963,A -85,B 0,C 180,E1 -5304.465,E2 -5304.465} C_VEL
LIN {X 0,Y 510.057,Z 636.953,A -85,B 0,C 180,E1 -5307.631,E2 -5307.631} C_VEL
LIN {X 0,Y 510.067,Z 636.952,A -85,B 0,C 180,E1 -5310.79,E2 -5310.79} C_VEL
LIN {X 0,Y 509.958,Z 636.965,A -85,B 0,C 180,E1 -5313.16,E2 -5313.16} C_VEL
LIN {X 0,Y 509.955,Z 636.963,A -85,B 0,C 180,E1 -5316.33,E2 -5316.33} C_VEL
LIN {X 0,Y 509.919,Z 636.971,A -85,B 0,C 180,E1 -5318.721,E2 -5318.721} C_VEL
LIN {X 0,Y 509.954,Z 636.963,A -85,B 0,C 180,E1 -5321.931,E2 -5321.931} C_VEL
LIN {X 0,Y 509.896,Z 636.974,A -85,B 0,C 180,E1 -5325.242,E2 -5325.242} C_VEL
LIN {X 0,Y 509.891,Z 636.975,A -85,B 0,C 180,E1 -5328.001,E2 -5328.001} C_VEL
LIN {X 0,Y 509.852,Z 636.978,A -85,B 0,C 180,E1 -5331.002,E2 -5331.002} C_VEL
LIN {X 0,Y 509.887,Z 636.975,A -85,B 0,C 180,E1 -5334.535,E2 -5334.535} C_VEL
LIN {X 0,Y 509.892,Z 637.1,A -85,B 0,C 180,E1 -5334.686,E2 -5334.686} C_VEL
LIN {X 0,Y 511.533,Z 643.752,A -85,B 0,C 180,E1 -5335.05,E2 -5335.05} C_VEL
LIN {X 0,Y 511.269,Z 656.235,A -85,B 0,C 180,E1 -5335.768,E2 -5335.768} C_VEL
LIN {X 0,Y 510.929,Z 667.536,A -85,B 0,C 180,E1 -5336.607,E2 -5336.607} C_VEL
LIN {X 0,Y 510.616,Z 677.8,A -85,B 0,C 180,E1 -5337.569,E2 -5337.569} C_VEL
LIN {X 0,Y 510.349,Z 687.051,A -85,B 0,C 180,E1 -5338.643,E2 -5338.643} C_VEL
LIN {X 0,Y 510.082,Z 694.947,A -85,B 0,C 180,E1 -5339.77,E2 -5339.77} C_VEL
LIN {X 0,Y 509.882,Z 701.699,A -85,B 0,C 180,E1 -5340.97,E2 -5340.97} C_VEL
LIN {X 0,Y 509.726,Z 706.657,A -85,B 0,C 180,E1 -5342.062,E2 -5342.062} C_VEL
LIN {X 0,Y 509.574,Z 711.649,A -85,B 0,C 180,E1 -5343.482,E2 -5343.482} C_VEL
LIN {X 0,Y 509.508,Z 714.166,A -85,B 0,C 180,E1 -5344.44,E2 -5344.44} C_VEL
LIN {X 0,Y 509.435,Z 716.274,A -85,B 0,C 180,E1 -5345.517,E2 -5345.517} C_VEL
LIN {X 0,Y 509.376,Z 717.835,A -85,B 0,C 180,E1 -5346.847,E2 -5346.847} C_VEL
LIN {X 0,Y 509.379,Z 718.253,A -85,B 0,C 180,E1 -5348.38,E2 -5348.38} C_VEL
LIN {X 0,Y 509.406,Z 717.739,A -85,B 0,C 180,E1 -5349.412,E2 -5349.412} C_VEL
LIN {X 0,Y 509.448,Z 716.244,A -85,B 0,C 180,E1 -5350.647,E2 -5350.647} C_VEL
LIN {X 0,Y 509.564,Z 713.81,A -85,B 0,C 180,E1 -5351.86,E2 -5351.86} C_VEL
LIN {X 0,Y 509.665,Z 710.467,A -85,B 0,C 180,E1 -5353.043,E2 -5353.043} C_VEL
LIN {X 0,Y 509.773,Z 705.323,A -85,B 0,C 180,E1 -5354.398,E2 -5354.398} C_VEL
LIN {X 0,Y 509.977,Z 699.918,A -85,B 0,C 180,E1 -5355.513,E2 -5355.513} C_VEL
LIN {X 0,Y 510.179,Z 693.424,A -85,B 0,C 180,E1 -5356.606,E2 -5356.606} C_VEL
LIN {X 0,Y 510.444,Z 685.431,A -85,B 0,C 180,E1 -5357.703,E2 -5357.703} C_VEL
LIN {X 0,Y 510.785,Z 675.426,A -85,B 0,C 180,E1 -5358.81,E2 -5358.81} C_VEL
LIN {X 0,Y 511.059,Z 664.933,A -85,B 0,C 180,E1 -5359.734,E2 -5359.734} C_VEL
LIN {X 0,Y 511.356,Z 653.706,A -85,B 0,C 180,E1 -5360.521,E2 -5360.521} C_VEL
LIN {X 0,Y 511.57,Z 643.989,A -85,B 0,C 180,E1 -5361.059,E2 -5361.059} C_VEL
LIN {X 0,Y 510.397,Z 639.008,A -85,B 0,C 180,E1 -5361.333,E2 -5361.333} C_VEL
LIN {X 0,Y 509.857,Z 636.979,A -85,B 0,C 180,E1 -5361.442,E2 -5361.442} C_VEL
LIN {X 0,Y 509.831,Z 636.975,A -85,B 0,C 180,E1 -5364.622,E2 -5364.622} C_VEL
LIN {X 0,Y 509.862,Z 636.979,A -85,B 0,C 180,E1 -5367.481,E2 -5367.481} C_VEL
LIN {X 0,Y 509.859,Z 636.971,A -85,B 0,C 180,E1 -5370.274,E2 -5370.274} C_VEL
LIN {X 0,Y 509.886,Z 636.968,A -85,B 0,C 180,E1 -5372.944,E2 -5372.944} C_VEL
LIN {X 0,Y 509.848,Z 636.978,A -85,B 0,C 180,E1 -5375.573,E2 -5375.573} C_VEL
LIN {X 0,Y 509.823,Z 636.979,A -85,B 0,C 180,E1 -5378.149,E2 -5378.149} C_VEL
LIN {X 0,Y 509.864,Z 636.97,A -85,B 0,C 180,E1 -5380.682,E2 -5380.682} C_VEL
LIN {X 0,Y 509.885,Z 636.968,A -85,B 0,C 180,E1 -5383.175,E2 -5383.175} C_VEL
LIN {X 0,Y 509.865,Z 636.976,A -85,B 0,C 180,E1 -5385.634,E2 -5385.634} C_VEL
LIN {X 0,Y 509.914,Z 636.961,A -85,B 0,C 180,E1 -5388.875,E2 -5388.875} C_VEL
LIN {X 0,Y 509.953,Z 636.962,A -85,B 0,C 180,E1 -5392.079,E2 -5392.079} C_VEL
LIN {X 0,Y 509.983,Z 636.957,A -85,B 0,C 180,E1 -5394.464,E2 -5394.464} C_VEL
LIN {X 0,Y 510.058,Z 636.945,A -85,B 0,C 180,E1 -5397.631,E2 -5397.631} C_VEL
LIN {X 0,Y 510.065,Z 636.941,A -85,B 0,C 180,E1 -5400.79,E2 -5400.79} C_VEL
LIN {X 0,Y 509.958,Z 636.957,A -85,B 0,C 180,E1 -5403.16,E2 -5403.16} C_VEL
LIN {X 0,Y 509.98,Z 636.962,A -85,B 0,C 180,E1 -5406.33,E2 -5406.33} C_VEL
LIN {X 0,Y 509.917,Z 636.962,A -85,B 0,C 180,E1 -5408.72,E2 -5408.72} C_VEL
LIN {X 0,Y 509.906,Z 636.969,A -85,B 0,C 180,E1 -5411.932,E2 -5411.932} C_VEL
LIN {X 0,Y 509.895,Z 636.965,A -85,B 0,C 180,E1 -5415.242,E2 -5415.242} C_VEL
LIN {X 0,Y 509.883,Z 636.97,A -85,B 0,C 180,E1 -5417.999,E2 -5417.999} C_VEL
LIN {X 0,Y 509.851,Z 636.972,A -85,B 0,C 180,E1 -5421.002,E2 -5421.002} C_VEL
LIN {X 0,Y 509.867,Z 636.978,A -85,B 0,C 180,E1 -5424.426,E2 -5424.426} C_VEL
LIN {X 0,Y 509.887,Z 636.968,A -85,B 0,C 180,E1 -5427.056,E2 -5427.056} C_VEL
LIN {X 0,Y 509.859,Z 636.971,A -85,B 0,C 180,E1 -5429.751,E2 -5429.751} C_VEL
LIN {X 0,Y 509.875,Z 636.975,A -85,B 0,C 180,E1 -5432.774,E2 -5432.774} C_VEL
LIN {X 0,Y 509.828,Z 636.975,A -85,B 0,C 180,E1 -5435.579,E2 -5435.579} C_VEL
LIN {X 0,Y 509.853,Z 636.978,A -85,B 0,C 180,E1 -5438.338,E2 -5438.338} C_VEL
LIN {X 0,Y 509.866,Z 636.971,A -85,B 0,C 180,E1 -5441.425,E2 -5441.425} C_VEL
LIN {X 0,Y 509.859,Z 636.978,A -85,B 0,C 180,E1 -5444.668,E2 -5444.668} C_VEL
LIN {X 0,Y 509.858,Z 636.976,A -85,B 0,C 180,E1 -5448.103,E2 -5448.103} C_VEL
LIN {X 0,Y 509.852,Z 637.01,A -85,B 0,C 180,E1 -5451.157,E2 -5451.157} C_VEL
LIN {X 0,Y 511.553,Z 645.598,A -85,B 0,C 180,E1 -5453.354,E2 -5453.354} C_VEL
LIN {X 0,Y 511.712,Z 651.604,A -85,B 0,C 180,E1 -5454.771,E2 -5454.771} C_VEL
LIN {X 0,Y 511.387,Z 665.132,A -85,B 0,C 180,E1 -5457.823,E2 -5457.823} C_VEL
LIN {X 0,Y 511.129,Z 678.817,A -85,B 0,C 180,E1 -5460.782,E2 -5460.782} C_VEL
LIN {X 0,Y 510.88,Z 693.571,A -85,B 0,C 180,E1 -5463.882,E2 -5463.882} C_VEL
LIN {X 0,Y 510.598,Z 708.238,A -85,B 0,C 180,E1 -5466.904,E2 -5466.904} C_VEL
LIN {X 0,Y 510.333,Z 724.278,A -85,B 0,C 180,E1 -5470.072,E2 -5470.072} C_VEL
LIN {X 0,Y 510.076,Z 739.051,A -85,B 0,C 180,E1 -5472.975,E2 -5472.975} C_VEL
LIN {X 0,Y 509.845,Z 753.815,A -85,B 0,C 180,E1 -5475.869,E2 -5475.869} C_VEL
LIN {X 0,Y 511.659,Z 766.193,A -85,B 0,C 180,E1 -5476.167,E2 -5476.167} C_VEL
LIN {X 0,Y 511.385,Z 779.358,A -85,B 0,C 180,E1 -5476.59,E2 -5476.59} C_VEL
LIN {X 0,Y 511.107,Z 790.466,A -85,B 0,C 180,E1 -5477.088,E2 -5477.088} C_VEL
LIN {X 0,Y 510.828,Z 801.915,A -85,B 0,C 180,E1 -5477.76,E2 -5477.76} C_VEL
LIN {X 0,Y 510.551,Z 812.913,A -85,B 0,C 180,E1 -5478.587,E2 -5478.587} C_VEL
LIN {X 0,Y 510.173,Z 822.593,A -85,B 0,C 180,E1 -5479.483,E2 -5479.483} C_VEL
LIN {X 0,Y 509.887,Z 831.41,A -85,B 0,C 180,E1 -5480.479,E2 -5480.479} C_VEL
LIN {X 0,Y 509.625,Z 840.002,A -85,B 0,C 180,E1 -5481.674,E2 -5481.674} C_VEL
LIN {X 0,Y 509.423,Z 846.867,A -85,B 0,C 180,E1 -5482.867,E2 -5482.867} C_VEL
LIN {X 0,Y 509.369,Z 852.363,A -85,B 0,C 180,E1 -5484.06,E2 -5484.06} C_VEL
LIN {X 0,Y 509.189,Z 856.675,A -85,B 0,C 180,E1 -5485.249,E2 -5485.249} C_VEL
LIN {X 0,Y 509.254,Z 858.959,A -85,B 0,C 180,E1 -5486.043,E2 -5486.043} C_VEL
LIN {X 0,Y 509.201,Z 860.809,A -85,B 0,C 180,E1 -5486.835,E2 -5486.835} C_VEL
LIN {X 0,Y 509.16,Z 862.195,A -85,B 0,C 180,E1 -5487.626,E2 -5487.626} C_VEL
LIN {X 0,Y 509.073,Z 863.786,A -85,B 0,C 180,E1 -5489.209,E2 -5489.209} C_VEL
LIN {X 0,Y 509.065,Z 864,A -85,B 0,C 180,E1 -5490,E2 -5490} C_VEL
LIN {X 0,Y 509.112,Z 863.182,A -85,B 0,C 180,E1 -5491.582,E2 -5491.582} C_VEL
LIN {X 0,Y 509.16,Z 862.194,A -85,B 0,C 180,E1 -5492.373,E2 -5492.373} C_VEL
LIN {X 0,Y 509.201,Z 860.808,A -85,B 0,C 180,E1 -5493.164,E2 -5493.164} C_VEL
LIN {X 0,Y 509.234,Z 857.895,A -85,B 0,C 180,E1 -5494.353,E2 -5494.353} C_VEL
LIN {X 0,Y 509.344,Z 853.951,A -85,B 0,C 180,E1 -5495.542,E2 -5495.542} C_VEL
LIN {X 0,Y 509.41,Z 848.283,A -85,B 0,C 180,E1 -5496.853,E2 -5496.853} C_VEL
LIN {X 0,Y 509.585,Z 841.238,A -85,B 0,C 180,E1 -5498.126,E2 -5498.126} C_VEL
LIN {X 0,Y 509.845,Z 832.996,A -85,B 0,C 180,E1 -5499.321,E2 -5499.321} C_VEL
LIN {X 0,Y 510.068,Z 824.544,A -85,B 0,C 180,E1 -5500.318,E2 -5500.318} C_VEL
LIN {X 0,Y 510.461,Z 814.097,A -85,B 0,C 180,E1 -5501.314,E2 -5501.314} C_VEL
LIN {X 0,Y 510.768,Z 803.23,A -85,B 0,C 180,E1 -5502.149,E2 -5502.149} C_VEL
LIN {X 0,Y 511.071,Z 792.41,A -85,B 0,C 180,E1 -5502.811,E2 -5502.811} C_VEL
LIN {X 0,Y 511.379,Z 780.706,A -85,B 0,C 180,E1 -5503.359,E2 -5503.359} C_VEL
LIN {X 0,Y 511.618,Z 768.089,A -85,B 0,C 180,E1 -5503.783,E2 -5503.783} C_VEL
LIN {X 0,Y 511.252,Z 763.092,A -85,B 0,C 180,E1 -5503.919,E2 -5503.919} C_VEL
LIN {X 0,Y 509.827,Z 753.766,A -85,B 0,C 180,E1 -5504.147,E2 -5504.147} C_VEL
LIN {X 0,Y 510.098,Z 738.216,A -85,B 0,C 180,E1 -5507.23,E2 -5507.23} C_VEL
LIN {X 0,Y 510.35,Z 723.621,A -85,B 0,C 180,E1 -5510.137,E2 -5510.137} C_VEL
LIN {X 0,Y 510.665,Z 709.089,A -85,B 0,C 180,E1 -5513.092,E2 -5513.092} C_VEL
LIN {X 0,Y 511.021,Z 693.352,A -85,B 0,C 180,E1 -5516.37,E2 -5516.37} C_VEL
LIN {X 0,Y 511.334,Z 679.097,A -85,B 0,C 180,E1 -5519.429,E2 -5519.429} C_VEL
LIN {X 0,Y 511.624,Z 667.713,A -85,B 0,C 180,E1 -5521.943,E2 -5521.943} C_VEL
LIN {X 0,Y 511.977,Z 655.066,A -85,B 0,C 180,E1 -5524.826,E2 -5524.826} C_VEL
LIN {X 0,Y 512.084,Z 648.336,A -85,B 0,C 180,E1 -5526.406,E2 -5526.406} C_VEL
LIN {X 0,Y 510.253,Z 638.988,A -85,B 0,C 180,E1 -5528.805,E2 -5528.805} C_VEL
LIN {X 0,Y 509.847,Z 636.979,A -85,B 0,C 180,E1 -5529.351,E2 -5529.351} C_VEL
LIN {X 0,Y 509.831,Z 636.981,A -85,B 0,C 180,E1 -5532.489,E2 -5532.489} C_VEL
LIN {X 0,Y 509.854,Z 636.974,A -85,B 0,C 180,E1 -5535.331,E2 -5535.331} C_VEL
LIN {X 0,Y 509.863,Z 636.977,A -85,B 0,C 180,E1 -5538.575,E2 -5538.575} C_VEL
LIN {X 0,Y 509.857,Z 636.973,A -85,B 0,C 180,E1 -5541.662,E2 -5541.662} C_VEL
LIN {X 0,Y 509.84,Z 636.974,A -85,B 0,C 180,E1 -5544.622,E2 -5544.622} C_VEL
LIN {X 0,Y 509.86,Z 636.973,A -85,B 0,C 180,E1 -5547.481,E2 -5547.481} C_VEL
LIN {X 0,Y 509.878,Z 636.971,A -85,B 0,C 180,E1 -5550.268,E2 -5550.268} C_VEL
LIN {X 0,Y 509.883,Z 636.969,A -85,B 0,C 180,E1 -5552.944,E2 -5552.944} C_VEL
LIN {X 0,Y 509.866,Z 636.978,A -85,B 0,C 180,E1 -5555.574,E2 -5555.574} C_VEL
LIN {X 0,Y 509.818,Z 636.977,A -85,B 0,C 180,E1 -5558.148,E2 -5558.148} C_VEL
LIN {X 0,Y 509.861,Z 636.972,A -85,B 0,C 180,E1 -5560.681,E2 -5560.681} C_VEL
LIN {X 0,Y 509.88,Z 636.975,A -85,B 0,C 180,E1 -5563.174,E2 -5563.174} C_VEL
LIN {X 0,Y 509.859,Z 636.973,A -85,B 0,C 180,E1 -5565.634,E2 -5565.634} C_VEL
LIN {X 0,Y 509.921,Z 636.969,A -85,B 0,C 180,E1 -5568.875,E2 -5568.875} C_VEL
LIN {X 0,Y 509.947,Z 636.963,A -85,B 0,C 180,E1 -5572.078,E2 -5572.078} C_VEL
LIN {X 0,Y 509.977,Z 636.963,A -85,B 0,C 180,E1 -5574.464,E2 -5574.464} C_VEL
LIN {X 0,Y 510.049,Z 636.949,A -85,B 0,C 180,E1 -5577.631,E2 -5577.631} C_VEL
LIN {X 0,Y 510.059,Z 636.951,A -85,B 0,C 180,E1 -5580.789,E2 -5580.789} C_VEL
LIN {X 0,Y 509.955,Z 636.964,A -85,B 0,C 180,E1 -5583.16,E2 -5583.16} C_VEL
LIN {X 0,Y 509.901,Z 637.059,A -85,B 0,C 180,E1 -5584.248,E2 -5584.248} C_VEL
LIN {X 0,Y 510.555,Z 642.333,A -85,B 0,C 180,E1 -5585.529,E2 -5585.529} C_VEL
LIN {X 0,Y 510.675,Z 653.758,A -85,B 0,C 180,E1 -5588.308,E2 -5588.308} C_VEL
LIN {X 0,Y 510.657,Z 666.656,A -85,B 0,C 180,E1 -5591.511,E2 -5591.511} C_VEL
LIN {X 0,Y 510.519,Z 679.454,A -85,B 0,C 180,E1 -5594.754,E2 -5594.754} C_VEL
LIN {X 0,Y 510.332,Z 690.556,A -85,B 0,C 180,E1 -5597.636,E2 -5597.636} C_VEL
LIN {X 0,Y 510.151,Z 701.581,A -85,B 0,C 180,E1 -5600.483,E2 -5600.483} C_VEL
LIN {X 0,Y 509.914,Z 713.255,A -85,B 0,C 180,E1 -5603.559,E2 -5603.559} C_VEL
LIN {X 0,Y 509.695,Z 724.831,A -85,B 0,C 180,E1 -5606.663,E2 -5606.663} C_VEL
LIN {X 0,Y 509.699,Z 725.769,A -85,B 0,C 180,E1 -5606.915,E2 -5606.915} C_VEL
LIN {X 0,Y 511.591,Z 738.864,A -85,B 0,C 180,E1 -5607.276,E2 -5607.276} C_VEL
LIN {X 0,Y 511.321,Z 752.322,A -85,B 0,C 180,E1 -5607.749,E2 -5607.749} C_VEL
LIN {X 0,Y 510.989,Z 764.954,A -85,B 0,C 180,E1 -5608.373,E2 -5608.373} C_VEL
LIN {X 0,Y 510.654,Z 776.616,A -85,B 0,C 180,E1 -5609.134,E2 -5609.134} C_VEL
LIN {X 0,Y 510.343,Z 786.666,A -85,B 0,C 180,E1 -5609.954,E2 -5609.954} C_VEL
LIN {X 0,Y 510.024,Z 795.81,A -85,B 0,C 180,E1 -5610.864,E2 -5610.864} C_VEL
LIN {X 0,Y 509.792,Z 803.767,A -85,B 0,C 180,E1 -5611.824,E2 -5611.824} C_VEL
LIN {X 0,Y 509.568,Z 812.18,A -85,B 0,C 180,E1 -5613.074,E2 -5613.074} C_VEL
LIN {X 0,Y 509.423,Z 817.97,A -85,B 0,C 180,E1 -5614.132,E2 -5614.132} C_VEL
LIN {X 0,Y 509.275,Z 823.921,A -85,B 0,C 180,E1 -5615.493,E2 -5615.493} C_VEL
LIN {X 0,Y 509.196,Z 828.25,A -85,B 0,C 180,E1 -5616.821,E2 -5616.821} C_VEL
LIN {X 0,Y 509.115,Z 831.236,A -85,B 0,C 180,E1 -5618.109,E2 -5618.109} C_VEL
LIN {X 0,Y 509.068,Z 833.143,A -85,B 0,C 180,E1 -5619.424,E2 -5619.424} C_VEL
LIN {X 0,Y 509.046,Z 833.917,A -85,B 0,C 180,E1 -5620.595,E2 -5620.595} C_VEL
LIN {X 0,Y 509.038,Z 833.809,A -85,B 0,C 180,E1 -5621.795,E2 -5621.795} C_VEL
LIN {X 0,Y 509.081,Z 832.818,A -85,B 0,C 180,E1 -5622.974,E2 -5622.974} C_VEL
LIN {X 0,Y 509.136,Z 830.97,A -85,B 0,C 180,E1 -5624.128,E2 -5624.128} C_VEL
LIN {X 0,Y 509.178,Z 829.422,A -85,B 0,C 180,E1 -5624.82,E2 -5624.82} C_VEL
LIN {X 0,Y 508.535,Z 827.754,A -85,B 0,C 180,E1 -5625.452,E2 -5625.452} C_VEL
LIN {X 0,Y 505.766,Z 824.529,A -85,B 0,C 180,E1 -5626.467,E2 -5626.467} C_VEL
LIN {X 0,Y 502.975,Z 820.728,A -85,B 0,C 180,E1 -5627.462,E2 -5627.462} C_VEL
LIN {X 0,Y 502.307,Z 818.02,A -85,B 0,C 180,E1 -5628.06,E2 -5628.06} C_VEL
LIN {X 0,Y 502.505,Z 811.401,A -85,B 0,C 180,E1 -5629.275,E2 -5629.275} C_VEL
LIN {X 0,Y 502.79,Z 803.033,A -85,B 0,C 180,E1 -5630.507,E2 -5630.507} C_VEL
LIN {X 0,Y 503.143,Z 793.52,A -85,B 0,C 180,E1 -5631.626,E2 -5631.626} C_VEL
LIN {X 0,Y 503.517,Z 783.21,A -85,B 0,C 180,E1 -5632.609,E2 -5632.609} C_VEL
LIN {X 0,Y 503.837,Z 771.827,A -85,B 0,C 180,E1 -5633.47,E2 -5633.47} C_VEL
LIN {X 0,Y 504.249,Z 759.946,A -85,B 0,C 180,E1 -5634.171,E2 -5634.171} C_VEL
LIN {X 0,Y 504.498,Z 748.615,A -85,B 0,C 180,E1 -5634.682,E2 -5634.682} C_VEL
LIN {X 0,Y 504.636,Z 738.227,A -85,B 0,C 180,E1 -5635.029,E2 -5635.029} C_VEL
LIN {X 0,Y 502.621,Z 725.907,A -85,B 0,C 180,E1 -5635.375,E2 -5635.375} C_VEL
LIN {X 0,Y 502.849,Z 714.297,A -85,B 0,C 180,E1 -5638.491,E2 -5638.491} C_VEL
LIN {X 0,Y 503.143,Z 702.496,A -85,B 0,C 180,E1 -5641.647,E2 -5641.647} C_VEL
LIN {X 0,Y 503.427,Z 690.69,A -85,B 0,C 180,E1 -5644.801,E2 -5644.801} C_VEL
LIN {X 0,Y 503.616,Z 679.213,A -85,B 0,C 180,E1 -5647.866,E2 -5647.866} C_VEL
LIN {X 0,Y 503.811,Z 669.582,A -85,B 0,C 180,E1 -5650.441,E2 -5650.441} C_VEL
LIN {X 0,Y 503.919,Z 658.512,A -85,B 0,C 180,E1 -5653.388,E2 -5653.388} C_VEL
LIN {X 0,Y 503.999,Z 647.589,A -85,B 0,C 180,E1 -5656.288,E2 -5656.288} C_VEL
LIN {X 0,Y 503.552,Z 641.544,A -85,B 0,C 180,E1 -5657.916,E2 -5657.916} C_VEL
LIN {X 0,Y 502.888,Z 637.844,A -85,B 0,C 180,E1 -5658.973,E2 -5658.973} C_VEL
LIN {X 0,Y 502.903,Z 637.842,A -85,B 0,C 180,E1 -5661.967,E2 -5661.967} C_VEL
LIN {X 0,Y 502.94,Z 637.84,A -85,B 0,C 180,E1 -5664.387,E2 -5664.387} C_VEL
LIN {X 0,Y 503.027,Z 637.828,A -85,B 0,C 180,E1 -5667.598,E2 -5667.598} C_VEL
LIN {X 0,Y 503.03,Z 637.826,A -85,B 0,C 180,E1 -5670,E2 -5670} C_VEL
LIN {X 0,Y 503.027,Z 637.828,A -85,B 0,C 180,E1 -5672.403,E2 -5672.403} C_VEL
LIN {X 0,Y 502.935,Z 637.838,A -85,B 0,C 180,E1 -5675.614,E2 -5675.614} C_VEL
LIN {X 0,Y 502.904,Z 637.842,A -85,B 0,C 180,E1 -5678.034,E2 -5678.034} C_VEL
LIN {X 0,Y 502.894,Z 637.845,A -85,B 0,C 180,E1 -5681.283,E2 -5681.283} C_VEL
LIN {X 0,Y 502.848,Z 637.849,A -85,B 0,C 180,E1 -5684.571,E2 -5684.571} C_VEL
LIN {X 0,Y 502.864,Z 637.85,A -85,B 0,C 180,E1 -5687.907,E2 -5687.907} C_VEL
LIN {X 0,Y 502.831,Z 637.855,A -85,B 0,C 180,E1 -5690.536,E2 -5690.536} C_VEL
LIN {X 0,Y 502.794,Z 637.857,A -85,B 0,C 180,E1 -5693.914,E2 -5693.914} C_VEL
LIN {X 0,Y 502.848,Z 637.852,A -85,B 0,C 180,E1 -5694.484,E2 -5694.484} C_VEL
LIN {X 0,Y 504.477,Z 643.757,A -85,B 0,C 180,E1 -5694.816,E2 -5694.816} C_VEL
LIN {X 0,Y 504.52,Z 653.497,A -85,B 0,C 180,E1 -5695.363,E2 -5695.363} C_VEL
LIN {X 0,Y 504.194,Z 664.854,A -85,B 0,C 180,E1 -5696.157,E2 -5696.157} C_VEL
LIN {X 0,Y 503.864,Z 675.119,A -85,B 0,C 180,E1 -5697.055,E2 -5697.055} C_VEL
LIN {X 0,Y 503.52,Z 684.805,A -85,B 0,C 180,E1 -5698.104,E2 -5698.104} C_VEL
LIN {X 0,Y 503.236,Z 693.365,A -85,B 0,C 180,E1 -5699.262,E2 -5699.262} C_VEL
LIN {X 0,Y 502.986,Z 700.386,A -85,B 0,C 180,E1 -5700.432,E2 -5700.432} C_VEL
LIN {X 0,Y 502.778,Z 706.711,A -85,B 0,C 180,E1 -5701.752,E2 -5701.752} C_VEL
LIN {X 0,Y 502.632,Z 711.504,A -85,B 0,C 180,E1 -5703.046,E2 -5703.046} C_VEL
LIN {X 0,Y 502.499,Z 715.174,A -85,B 0,C 180,E1 -5704.393,E2 -5704.393} C_VEL
LIN {X 0,Y 502.409,Z 717.986,A -85,B 0,C 180,E1 -5705.982,E2 -5705.982} C_VEL
LIN {X 0,Y 502.365,Z 719.023,A -85,B 0,C 180,E1 -5707.116,E2 -5707.116} C_VEL
LIN {X 0,Y 502.371,Z 719.266,A -85,B 0,C 180,E1 -5708.425,E2 -5708.425} C_VEL
LIN {X 0,Y 502.413,Z 718.145,A -85,B 0,C 180,E1 -5710.051,E2 -5710.051} C_VEL
LIN {X 0,Y 502.515,Z 715.485,A -85,B 0,C 180,E1 -5711.63,E2 -5711.63} C_VEL
LIN {X 0,Y 502.634,Z 712.764,A -85,B 0,C 180,E1 -5712.698,E2 -5712.698} C_VEL
LIN {X 0,Y 502.744,Z 708.066,A -85,B 0,C 180,E1 -5714.077,E2 -5714.077} C_VEL
LIN {X 0,Y 502.988,Z 701.882,A -85,B 0,C 180,E1 -5715.447,E2 -5715.447} C_VEL
LIN {X 0,Y 503.186,Z 695.448,A -85,B 0,C 180,E1 -5716.576,E2 -5716.576} C_VEL
LIN {X 0,Y 503.5,Z 687.443,A -85,B 0,C 180,E1 -5717.714,E2 -5717.714} C_VEL
LIN {X 0,Y 503.791,Z 678.956,A -85,B 0,C 180,E1 -5718.701,E2 -5718.701} C_VEL
LIN {X 0,Y 504.128,Z 669.638,A -85,B 0,C 180,E1 -5719.59,E2 -5719.59} C_VEL
LIN {X 0,Y 504.466,Z 659.122,A -85,B 0,C 180,E1 -5720.404,E2 -5720.404} C_VEL
LIN {X 0,Y 504.709,Z 648.224,A -85,B 0,C 180,E1 -5721.071,E2 -5721.071} C_VEL
LIN {X 0,Y 504.505,Z 643.786,A -85,B 0,C 180,E1 -5721.31,E2 -5721.31} C_VEL
LIN {X 0,Y 502.826,Z 637.853,A -85,B 0,C 180,E1 -5721.651,E2 -5721.651} C_VEL
LIN {X 0,Y 502.8,Z 637.853,A -85,B 0,C 180,E1 -5725.034,E2 -5725.034} C_VEL
LIN {X 0,Y 502.784,Z 637.857,A -85,B 0,C 180,E1 -5727.915,E2 -5727.915} C_VEL
LIN {X 0,Y 502.825,Z 637.846,A -85,B 0,C 180,E1 -5730.712,E2 -5730.712} C_VEL
LIN {X 0,Y 502.864,Z 637.847,A -85,B 0,C 180,E1 -5733.439,E2 -5733.439} C_VEL
LIN {X 0,Y 502.776,Z 637.854,A -85,B 0,C 180,E1 -5736.086,E2 -5736.086} C_VEL
LIN {X 0,Y 502.784,Z 637.853,A -85,B 0,C 180,E1 -5738.689,E2 -5738.689} C_VEL
LIN {X 0,Y 502.831,Z 637.848,A -85,B 0,C 180,E1 -5741.248,E2 -5741.248} C_VEL
LIN {X 0,Y 502.823,Z 637.854,A -85,B 0,C 180,E1 -5743.767,E2 -5743.767} C_VEL
LIN {X 0,Y 502.832,Z 637.85,A -85,B 0,C 180,E1 -5746.255,E2 -5746.255} C_VEL
LIN {X 0,Y 502.878,Z 637.838,A -85,B 0,C 180,E1 -5748.717,E2 -5748.717} C_VEL
LIN {X 0,Y 502.903,Z 637.841,A -85,B 0,C 180,E1 -5751.967,E2 -5751.967} C_VEL
LIN {X 0,Y 502.939,Z 637.835,A -85,B 0,C 180,E1 -5754.387,E2 -5754.387} C_VEL
LIN {X 0,Y 503.027,Z 637.821,A -85,B 0,C 180,E1 -5757.598,E2 -5757.598} C_VEL
LIN {X 0,Y 503.029,Z 637.827,A -85,B 0,C 180,E1 -5760,E2 -5760} C_VEL
LIN {X 0,Y 503.027,Z 637.825,A -85,B 0,C 180,E1 -5762.402,E2 -5762.402} C_VEL
LIN {X 0,Y 502.939,Z 637.83,A -85,B 0,C 180,E1 -5765.614,E2 -5765.614} C_VEL
LIN {X 0,Y 502.903,Z 637.843,A -85,B 0,C 180,E1 -5768.033,E2 -5768.033} C_VEL
LIN {X 0,Y 502.879,Z 637.84,A -85,B 0,C 180,E1 -5771.283,E2 -5771.283} C_VEL
LIN {X 0,Y 502.847,Z 637.848,A -85,B 0,C 180,E1 -5774.571,E2 -5774.571} C_VEL
LIN {X 0,Y 502.857,Z 637.844,A -85,B 0,C 180,E1 -5777.907,E2 -5777.907} C_VEL
LIN {X 0,Y 502.83,Z 637.852,A -85,B 0,C 180,E1 -5780.536,E2 -5780.536} C_VEL
LIN {X 0,Y 502.793,Z 637.85,A -85,B 0,C 180,E1 -5783.041,E2 -5783.041} C_VEL
LIN {X 0,Y 502.842,Z 637.844,A -85,B 0,C 180,E1 -5785.676,E2 -5785.676} C_VEL
LIN {X 0,Y 502.842,Z 637.851,A -85,B 0,C 180,E1 -5788.373,E2 -5788.373} C_VEL
LIN {X 0,Y 502.794,Z 637.851,A -85,B 0,C 180,E1 -5791.499,E2 -5791.499} C_VEL
LIN {X 0,Y 502.805,Z 637.852,A -85,B 0,C 180,E1 -5793.994,E2 -5793.994} C_VEL
LIN {X 0,Y 502.78,Z 637.856,A -85,B 0,C 180,E1 -5797.178,E2 -5797.178} C_VEL
LIN {X 0,Y 502.793,Z 637.853,A -85,B 0,C 180,E1 -5800.015,E2 -5800.015} C_VEL
LIN {X 0,Y 502.805,Z 637.853,A -85,B 0,C 180,E1 -5802.199,E2 -5802.199} C_VEL
LIN {X 0,Y 502.803,Z 637.852,A -85,B 0,C 180,E1 -5805.468,E2 -5805.468} C_VEL
LIN {X 0,Y 502.822,Z 637.86,A -85,B 0,C 180,E1 -5808.934,E2 -5808.934} C_VEL
LIN {X 0,Y 502.802,Z 637.874,A -85,B 0,C 180,E1 -5810.895,E2 -5810.895} C_VEL
LIN {X 0,Y 504.559,Z 646.712,A -85,B 0,C 180,E1 -5813.205,E2 -5813.205} C_VEL
LIN {X 0,Y 504.824,Z 651.919,A -85,B 0,C 180,E1 -5814.463,E2 -5814.463} C_VEL
LIN {X 0,Y 504.41,Z 665.362,A -85,B 0,C 180,E1 -5817.559,E2 -5817.559} C_VEL
LIN {X 0,Y 504.132,Z 677.912,A -85,B 0,C 180,E1 -5820.337,E2 -5820.337} C_VEL
LIN {X 0,Y 503.874,Z 691.349,A -85,B 0,C 180,E1 -5823.211,E2 -5823.211} C_VEL
LIN {X 0,Y 503.591,Z 705.221,A -85,B 0,C 180,E1 -5826.126,E2 -5826.126} C_VEL
LIN {X 0,Y 503.33,Z 719.665,A -85,B 0,C 180,E1 -5829.061,E2 -5829.061} C_VEL
LIN {X 0,Y 503.06,Z 735.949,A -85,B 0,C 180,E1 -5832.31,E2 -5832.31} C_VEL
LIN {X 0,Y 502.793,Z 751.617,A -85,B 0,C 180,E1 -5835.427,E2 -5835.427} C_VEL
LIN {X 0,Y 502.779,Z 752.77,A -85,B 0,C 180,E1 -5835.66,E2 -5835.66} C_VEL
LIN {X 0,Y 504.678,Z 766.895,A -85,B 0,C 180,E1 -5836.023,E2 -5836.023} C_VEL
LIN {X 0,Y 504.398,Z 779.531,A -85,B 0,C 180,E1 -5836.452,E2 -5836.452} C_VEL
LIN {X 0,Y 504.075,Z 791.354,A -85,B 0,C 180,E1 -5837.007,E2 -5837.007} C_VEL
LIN {X 0,Y 503.801,Z 802.74,A -85,B 0,C 180,E1 -5837.705,E2 -5837.705} C_VEL
LIN {X 0,Y 503.441,Z 814.646,A -85,B 0,C 180,E1 -5838.627,E2 -5838.627} C_VEL
LIN {X 0,Y 503.062,Z 824.12,A -85,B 0,C 180,E1 -5839.536,E2 -5839.536} C_VEL
LIN {X 0,Y 502.794,Z 832.794,A -85,B 0,C 180,E1 -5840.547,E2 -5840.547} C_VEL
LIN {X 0,Y 502.543,Z 841.189,A -85,B 0,C 180,E1 -5841.758,E2 -5841.758} C_VEL
LIN {X 0,Y 502.346,Z 847.874,A -85,B 0,C 180,E1 -5842.968,E2 -5842.968} C_VEL
LIN {X 0,Y 502.26,Z 853.946,A -85,B 0,C 180,E1 -5844.379,E2 -5844.379} C_VEL
LIN {X 0,Y 502.129,Z 857.894,A -85,B 0,C 180,E1 -5845.585,E2 -5845.585} C_VEL
LIN {X 0,Y 502.121,Z 860.809,A -85,B 0,C 180,E1 -5846.79,E2 -5846.79} C_VEL
LIN {X 0,Y 502.035,Z 863.183,A -85,B 0,C 180,E1 -5848.395,E2 -5848.395} C_VEL
LIN {X 0,Y 501.98,Z 864,A -85,B 0,C 180,E1 -5850,E2 -5850} C_VEL
LIN {X 0,Y 502.035,Z 863.182,A -85,B 0,C 180,E1 -5851.604,E2 -5851.604} C_VEL
LIN {X 0,Y 502.121,Z 860.807,A -85,B 0,C 180,E1 -5853.209,E2 -5853.209} C_VEL
LIN {X 0,Y 502.128,Z 857.895,A -85,B 0,C 180,E1 -5854.415,E2 -5854.415} C_VEL
LIN {X 0,Y 502.259,Z 853.951,A -85,B 0,C 180,E1 -5855.621,E2 -5855.621} C_VEL
LIN {X 0,Y 502.335,Z 847.978,A -85,B 0,C 180,E1 -5857.011,E2 -5857.011} C_VEL
LIN {X 0,Y 502.542,Z 841.194,A -85,B 0,C 180,E1 -5858.241,E2 -5858.241} C_VEL
LIN {X 0,Y 502.79,Z 832.8,A -85,B 0,C 180,E1 -5859.453,E2 -5859.453} C_VEL
LIN {X 0,Y 503.06,Z 824.148,A -85,B 0,C 180,E1 -5860.463,E2 -5860.463} C_VEL
LIN {X 0,Y 503.454,Z 813.496,A -85,B 0,C 180,E1 -5861.473,E2 -5861.473} C_VEL
LIN {X 0,Y 503.761,Z 802.445,A -85,B 0,C 180,E1 -5862.321,E2 -5862.321} C_VEL
LIN {X 0,Y 504.075,Z 791.471,A -85,B 0,C 180,E1 -5862.992,E2 -5862.992} C_VEL
LIN {X 0,Y 504.397,Z 779.691,A -85,B 0,C 180,E1 -5863.547,E2 -5863.547} C_VEL
LIN {X 0,Y 504.651,Z 766.151,A -85,B 0,C 180,E1 -5864.002,E2 -5864.002} C_VEL
LIN {X 0,Y 502.839,Z 754.05,A -85,B 0,C 180,E1 -5864.312,E2 -5864.312} C_VEL
LIN {X 0,Y 502.782,Z 752.781,A -85,B 0,C 180,E1 -5864.365,E2 -5864.365} C_VEL
LIN {X 0,Y 503.072,Z 737.393,A -85,B 0,C 180,E1 -5867.479,E2 -5867.479} C_VEL
LIN {X 0,Y 503.338,Z 721.507,A -85,B 0,C 180,E1 -5870.689,E2 -5870.689} C_VEL
LIN {X 0,Y 503.654,Z 706.212,A -85,B 0,C 180,E1 -5873.87,E2 -5873.87} C_VEL
LIN {X 0,Y 504.042,Z 691.226,A -85,B 0,C 180,E1 -5877.063,E2 -5877.063} C_VEL
LIN {X 0,Y 504.428,Z 676.73,A -85,B 0,C 180,E1 -5880.251,E2 -5880.251} C_VEL
LIN {X 0,Y 504.859,Z 663.032,A -85,B 0,C 180,E1 -5883.358,E2 -5883.358} C_VEL
LIN {X 0,Y 505.266,Z 650.863,A -85,B 0,C 180,E1 -5886.22,E2 -5886.22} C_VEL
LIN {X 0,Y 504.163,Z 644.569,A -85,B 0,C 180,E1 -5887.832,E2 -5887.832} C_VEL
LIN {X 0,Y 502.791,Z 637.858,A -85,B 0,C 180,E1 -5889.638,E2 -5889.638} C_VEL
LIN {X 0,Y 502.8,Z 637.855,A -85,B 0,C 180,E1 -5892.198,E2 -5892.198} C_VEL
LIN {X 0,Y 502.798,Z 637.852,A -85,B 0,C 180,E1 -5895.468,E2 -5895.468} C_VEL
LIN {X 0,Y 502.827,Z 637.849,A -85,B 0,C 180,E1 -5897.864,E2 -5897.864} C_VEL
LIN {X 0,Y 502.821,Z 637.849,A -85,B 0,C 180,E1 -5901.026,E2 -5901.026} C_VEL
LIN {X 0,Y 502.781,Z 637.859,A -85,B 0,C 180,E1 -5904.167,E2 -5904.167} C_VEL
LIN {X 0,Y 502.829,Z 637.847,A -85,B 0,C 180,E1 -5906.993,E2 -5906.993} C_VEL
LIN {X 0,Y 502.827,Z 637.851,A -85,B 0,C 180,E1 -5910.061,E2 -5910.061} C_VEL
LIN {X 0,Y 502.831,Z 637.847,A -85,B 0,C 180,E1 -5912.533,E2 -5912.533} C_VEL
LIN {X 0,Y 502.824,Z 637.85,A -85,B 0,C 180,E1 -5915.298,E2 -5915.298} C_VEL
LIN {X 0,Y 502.78,Z 637.857,A -85,B 0,C 180,E1 -5917.826,E2 -5917.826} C_VEL
LIN {X 0,Y 502.821,Z 637.847,A -85,B 0,C 180,E1 -5920.4,E2 -5920.4} C_VEL
LIN {X 0,Y 502.829,Z 637.85,A -85,B 0,C 180,E1 -5922.931,E2 -5922.931} C_VEL
LIN {X 0,Y 502.84,Z 637.849,A -85,B 0,C 180,E1 -5925.429,E2 -5925.429} C_VEL
LIN {X 0,Y 502.89,Z 637.846,A -85,B 0,C 180,E1 -5928.717,E2 -5928.717} C_VEL
LIN {X 0,Y 502.897,Z 637.84,A -85,B 0,C 180,E1 -5931.966,E2 -5931.966} C_VEL
LIN {X 0,Y 502.933,Z 637.841,A -85,B 0,C 180,E1 -5934.386,E2 -5934.386} C_VEL
LIN {X 0,Y 503.019,Z 637.825,A -85,B 0,C 180,E1 -5937.598,E2 -5937.598} C_VEL
LIN {X 0,Y 503.021,Z 637.83,A -85,B 0,C 180,E1 -5940,E2 -5940} C_VEL
LIN {X 0,Y 503.02,Z 637.83,A -85,B 0,C 180,E1 -5942.402,E2 -5942.402} C_VEL
LIN {X 0,Y 502.87,Z 638.008,A -85,B 0,C 180,E1 -5944.107,E2 -5944.107} C_VEL
LIN {X 0,Y 503.538,Z 642.447,A -85,B 0,C 180,E1 -5945.205,E2 -5945.205} C_VEL
LIN {X 0,Y 503.691,Z 653.967,A -85,B 0,C 180,E1 -5948.021,E2 -5948.021} C_VEL
LIN {X 0,Y 503.634,Z 665.343,A -85,B 0,C 180,E1 -5950.859,E2 -5950.859} C_VEL
LIN {X 0,Y 503.566,Z 675.022,A -85,B 0,C 180,E1 -5953.314,E2 -5953.314} C_VEL
LIN {X 0,Y 503.409,Z 686.266,A -85,B 0,C 180,E1 -5956.213,E2 -5956.213} C_VEL
LIN {X 0,Y 503.198,Z 697.452,A -85,B 0,C 180,E1 -5959.16,E2 -5959.16} C_VEL
LIN {X 0,Y 502.979,Z 708.904,A -85,B 0,C 180,E1 -5962.164,E2 -5962.164} C_VEL
LIN {X 0,Y 502.76,Z 720.465,A -85,B 0,C 180,E1 -5965.236,E2 -5965.236} C_VEL
LIN {X 0,Y 502.642,Z 725.91,A -85,B 0,C 180,E1 -5966.719,E2 -5966.719} C_VEL
LIN {X 0,Y 504.698,Z 738.687,A -85,B 0,C 180,E1 -5967.076,E2 -5967.076} C_VEL
LIN {X 0,Y 504.431,Z 751.867,A -85,B 0,C 180,E1 -5967.541,E2 -5967.541} C_VEL
LIN {X 0,Y 504.09,Z 763.864,A -85,B 0,C 180,E1 -5968.126,E2 -5968.126} C_VEL
LIN {X 0,Y 503.736,Z 775.018,A -85,B 0,C 180,E1 -5968.839,E2 -5968.839} C_VEL
LIN {X 0,Y 503.398,Z 785.829,A -85,B 0,C 180,E1 -5969.711,E2 -5969.711} C_VEL
LIN {X 0,Y 503.026,Z 795.402,A -85,B 0,C 180,E1 -5970.661,E2 -5970.661} C_VEL
LIN {X 0,Y 502.762,Z 804.381,A -85,B 0,C 180,E1 -5971.763,E2 -5971.763} C_VEL
LIN {X 0,Y 502.495,Z 812.834,A -85,B 0,C 180,E1 -5973.056,E2 -5973.056} C_VEL
LIN {X 0,Y 502.3,Z 819.602,A -85,B 0,C 180,E1 -5974.361,E2 -5974.361} C_VEL
LIN {X 0,Y 502.176,Z 825.092,A -85,B 0,C 180,E1 -5975.737,E2 -5975.737} C_VEL
LIN {X 0,Y 502.09,Z 829.075,A -85,B 0,C 180,E1 -5977.075,E2 -5977.075} C_VEL
LIN {X 0,Y 502.027,Z 831.784,A -85,B 0,C 180,E1 -5978.377,E2 -5978.377} C_VEL
LIN {X 0,Y 501.973,Z 833.381,A -85,B 0,C 180,E1 -5979.644,E2 -5979.644} C_VEL
LIN {X 0,Y 501.935,Z 833.985,A -85,B 0,C 180,E1 -5981.154,E2 -5981.154} C_VEL
LIN {X 0,Y 501.965,Z 833.562,A -85,B 0,C 180,E1 -5982.225,E2 -5982.225} C_VEL
LIN {X 0,Y 501.991,Z 832.386,A -85,B 0,C 180,E1 -5983.315,E2 -5983.315} C_VEL
LIN {X 0,Y 502.075,Z 829.515,A -85,B 0,C 180,E1 -5984.827,E2 -5984.827} C_VEL
LIN {X 0,Y 502.158,Z 825.787,A -85,B 0,C 180,E1 -5986.151,E2 -5986.151} C_VEL
LIN {X 0,Y 502.283,Z 820.436,A -85,B 0,C 180,E1 -5987.538,E2 -5987.538} C_VEL
LIN {X 0,Y 502.307,Z 818.02,A -85,B 0,C 180,E1 -5988.06,E2 -5988.06} C_VEL
LIN {X 0,Y 501.661,Z 815.122,A -85,B 0,C 180,E1 -5988.642,E2 -5988.642} C_VEL
LIN {X 0,Y 498.983,Z 810.055,A -85,B 0,C 180,E1 -5989.568,E2 -5989.568} C_VEL
LIN {X 0,Y 496.382,Z 804.429,A -85,B 0,C 180,E1 -5990.459,E2 -5990.459} C_VEL
LIN {X 0,Y 495.859,Z 800.575,A -85,B 0,C 180,E1 -5990.979,E2 -5990.979} C_VEL
LIN {X 0,Y 496.188,Z 791.895,A -85,B 0,C 180,E1 -5991.967,E2 -5991.967} C_VEL
LIN {X 0,Y 496.589,Z 781.845,A -85,B 0,C 180,E1 -5992.898,E2 -5992.898} C_VEL
LIN {X 0,Y 496.947,Z 770.873,A -85,B 0,C 180,E1 -5993.718,E2 -5993.718} C_VEL
LIN {X 0,Y 497.371,Z 759.029,A -85,B 0,C 180,E1 -5994.41,E2 -5994.41} C_VEL
LIN {X 0,Y 497.677,Z 746.011,A -85,B 0,C 180,E1 -5994.972,E2 -5994.972} C_VEL
LIN {X 0,Y 497.599,Z 738.026,A -85,B 0,C 180,E1 -5995.238,E2 -5995.238} C_VEL
LIN {X 0,Y 495.588,Z 726.095,A -85,B 0,C 180,E1 -5995.566,E2 -5995.566} C_VEL
LIN {X 0,Y 495.801,Z 715.749,A -85,B 0,C 180,E1 -5998.368,E2 -5998.368} C_VEL
LIN {X 0,Y 496.122,Z 704.346,A -85,B 0,C 180,E1 -6001.436,E2 -6001.436} C_VEL
LIN {X 0,Y 496.427,Z 691.603,A -85,B 0,C 180,E1 -6004.868,E2 -6004.868} C_VEL
LIN {X 0,Y 496.615,Z 680.082,A -85,B 0,C 180,E1 -6007.975,E2 -6007.975} C_VEL
LIN {X 0,Y 496.837,Z 670.377,A -85,B 0,C 180,E1 -6010.585,E2 -6010.585} C_VEL
LIN {X 0,Y 496.967,Z 659.259,A -85,B 0,C 180,E1 -6013.571,E2 -6013.571} C_VEL
LIN {X 0,Y 497.056,Z 648.27,A -85,B 0,C 180,E1 -6016.509,E2 -6016.509} C_VEL
LIN {X 0,Y 496.494,Z 642.248,A -85,B 0,C 180,E1 -6018.156,E2 -6018.156} C_VEL
LIN {X 0,Y 495.811,Z 638.725,A -85,B 0,C 180,E1 -6019.175,E2 -6019.175} C_VEL
LIN {X 0,Y 495.875,Z 638.718,A -85,B 0,C 180,E1 -6021.853,E2 -6021.853} C_VEL
LIN {X 0,Y 495.898,Z 638.718,A -85,B 0,C 180,E1 -6024.307,E2 -6024.307} C_VEL
LIN {X 0,Y 495.996,Z 638.704,A -85,B 0,C 180,E1 -6027.564,E2 -6027.564} C_VEL
LIN {X 0,Y 496.001,Z 638.702,A -85,B 0,C 180,E1 -6030,E2 -6030} C_VEL
LIN {X 0,Y 495.995,Z 638.703,A -85,B 0,C 180,E1 -6032.437,E2 -6032.437} C_VEL
LIN {X 0,Y 495.891,Z 638.716,A -85,B 0,C 180,E1 -6035.694,E2 -6035.694} C_VEL
LIN {X 0,Y 495.876,Z 638.717,A -85,B 0,C 180,E1 -6038.148,E2 -6038.148} C_VEL
LIN {X 0,Y 495.87,Z 638.721,A -85,B 0,C 180,E1 -6041.445,E2 -6041.445} C_VEL
LIN {X 0,Y 495.793,Z 638.727,A -85,B 0,C 180,E1 -6044.783,E2 -6044.783} C_VEL
LIN {X 0,Y 495.79,Z 638.728,A -85,B 0,C 180,E1 -6047.319,E2 -6047.319} C_VEL
LIN {X 0,Y 495.773,Z 638.731,A -85,B 0,C 180,E1 -6049.891,E2 -6049.891} C_VEL
LIN {X 0,Y 495.755,Z 638.734,A -85,B 0,C 180,E1 -6052.859,E2 -6052.859} C_VEL
LIN {X 0,Y 495.82,Z 638.834,A -85,B 0,C 180,E1 -6054.294,E2 -6054.294} C_VEL
LIN {X 0,Y 497.744,Z 646.07,A -85,B 0,C 180,E1 -6054.708,E2 -6054.708} C_VEL
LIN {X 0,Y 497.544,Z 658.554,A -85,B 0,C 180,E1 -6055.455,E2 -6055.455} C_VEL
LIN {X 0,Y 497.179,Z 669.878,A -85,B 0,C 180,E1 -6056.328,E2 -6056.328} C_VEL
LIN {X 0,Y 496.809,Z 680.604,A -85,B 0,C 180,E1 -6057.371,E2 -6057.371} C_VEL
LIN {X 0,Y 496.459,Z 690.122,A -85,B 0,C 180,E1 -6058.53,E2 -6058.53} C_VEL
LIN {X 0,Y 496.155,Z 697.981,A -85,B 0,C 180,E1 -6059.721,E2 -6059.721} C_VEL
LIN {X 0,Y 495.933,Z 704.334,A -85,B 0,C 180,E1 -6060.911,E2 -6060.911} C_VEL
LIN {X 0,Y 495.748,Z 709.511,A -85,B 0,C 180,E1 -6062.121,E2 -6062.121} C_VEL
LIN {X 0,Y 495.563,Z 714.28,A -85,B 0,C 180,E1 -6063.58,E2 -6063.58} C_VEL
LIN {X 0,Y 495.46,Z 716.827,A -85,B 0,C 180,E1 -6064.642,E2 -6064.642} C_VEL
LIN {X 0,Y 495.379,Z 719.104,A -85,B 0,C 180,E1 -6066.034,E2 -6066.034} C_VEL
LIN {X 0,Y 495.353,Z 720.249,A -85,B 0,C 180,E1 -6067.595,E2 -6067.595} C_VEL
LIN {X 0,Y 495.368,Z 720.222,A -85,B 0,C 180,E1 -6068.711,E2 -6068.711} C_VEL
LIN {X 0,Y 495.416,Z 719.269,A -85,B 0,C 180,E1 -6070,E2 -6070} C_VEL
LIN {X 0,Y 495.469,Z 717.393,A -85,B 0,C 180,E1 -6071.255,E2 -6071.255} C_VEL
LIN {X 0,Y 495.651,Z 713.424,A -85,B 0,C 180,E1 -6072.891,E2 -6072.891} C_VEL
LIN {X 0,Y 495.775,Z 709.724,A -85,B 0,C 180,E1 -6073.997,E2 -6073.997} C_VEL
LIN {X 0,Y 496.004,Z 703.92,A -85,B 0,C 180,E1 -6075.347,E2 -6075.347} C_VEL
LIN {X 0,Y 496.233,Z 697.796,A -85,B 0,C 180,E1 -6076.48,E2 -6076.48} C_VEL
LIN {X 0,Y 496.537,Z 690.126,A -85,B 0,C 180,E1 -6077.636,E2 -6077.636} C_VEL
LIN {X 0,Y 496.873,Z 680.783,A -85,B 0,C 180,E1 -6078.767,E2 -6078.767} C_VEL
LIN {X 0,Y 497.249,Z 670.72,A -85,B 0,C 180,E1 -6079.749,E2 -6079.749} C_VEL
LIN {X 0,Y 497.603,Z 660.713,A -85,B 0,C 180,E1 -6080.538,E2 -6080.538} C_VEL
LIN {X 0,Y 497.852,Z 650.184,A -85,B 0,C 180,E1 -6081.204,E2 -6081.204} C_VEL
LIN {X 0,Y 497.796,Z 645.84,A -85,B 0,C 180,E1 -6081.439,E2 -6081.439} C_VEL
LIN {X 0,Y 495.754,Z 638.733,A -85,B 0,C 180,E1 -6081.862,E2 -6081.862} C_VEL
LIN {X 0,Y 495.769,Z 638.731,A -85,B 0,C 180,E1 -6085.306,E2 -6085.306} C_VEL
LIN {X 0,Y 495.756,Z 638.73,A -85,B 0,C 180,E1 -6088.275,E2 -6088.275} C_VEL
LIN {X 0,Y 495.789,Z 638.729,A -85,B 0,C 180,E1 -6091.507,E2 -6091.507} C_VEL
LIN {X 0,Y 495.782,Z 638.729,A -85,B 0,C 180,E1 -6093.932,E2 -6093.932} C_VEL
LIN {X 0,Y 495.749,Z 638.73,A -85,B 0,C 180,E1 -6097.495,E2 -6097.495} C_VEL
LIN {X 0,Y 495.772,Z 638.73,A -85,B 0,C 180,E1 -6100.11,E2 -6100.11} C_VEL
LIN {X 0,Y 495.787,Z 638.723,A -85,B 0,C 180,E1 -6102.682,E2 -6102.682} C_VEL
LIN {X 0,Y 495.791,Z 638.725,A -85,B 0,C 180,E1 -6105.217,E2 -6105.217} C_VEL
LIN {X 0,Y 495.852,Z 638.714,A -85,B 0,C 180,E1 -6108.555,E2 -6108.555} C_VEL
LIN {X 0,Y 495.874,Z 638.718,A -85,B 0,C 180,E1 -6111.852,E2 -6111.852} C_VEL
LIN {X 0,Y 495.897,Z 638.714,A -85,B 0,C 180,E1 -6114.307,E2 -6114.307} C_VEL
LIN {X 0,Y 495.996,Z 638.696,A -85,B 0,C 180,E1 -6117.564,E2 -6117.564} C_VEL
LIN {X 0,Y 496,Z 638.702,A -85,B 0,C 180,E1 -6120,E2 -6120} C_VEL
LIN {X 0,Y 495.996,Z 638.701,A -85,B 0,C 180,E1 -6122.436,E2 -6122.436} C_VEL
LIN {X 0,Y 495.897,Z 638.708,A -85,B 0,C 180,E1 -6125.694,E2 -6125.694} C_VEL
LIN {X 0,Y 495.875,Z 638.718,A -85,B 0,C 180,E1 -6128.148,E2 -6128.148} C_VEL
LIN {X 0,Y 495.853,Z 638.715,A -85,B 0,C 180,E1 -6131.445,E2 -6131.445} C_VEL
LIN {X 0,Y 495.792,Z 638.725,A -85,B 0,C 180,E1 -6134.783,E2 -6134.783} C_VEL
LIN {X 0,Y 495.783,Z 638.722,A -85,B 0,C 180,E1 -6137.319,E2 -6137.319} C_VEL
LIN {X 0,Y 495.772,Z 638.726,A -85,B 0,C 180,E1 -6139.89,E2 -6139.89} C_VEL
LIN {X 0,Y 495.762,Z 638.728,A -85,B 0,C 180,E1 -6142.861,E2 -6142.861} C_VEL
LIN {X 0,Y 495.793,Z 638.725,A -85,B 0,C 180,E1 -6146.068,E2 -6146.068} C_VEL
LIN {X 0,Y 495.774,Z 638.729,A -85,B 0,C 180,E1 -6148.815,E2 -6148.815} C_VEL
LIN {X 0,Y 495.757,Z 638.728,A -85,B 0,C 180,E1 -6151.725,E2 -6151.725} C_VEL
LIN {X 0,Y 495.771,Z 638.733,A -85,B 0,C 180,E1 -6154.694,E2 -6154.694} C_VEL
LIN {X 0,Y 495.731,Z 638.732,A -85,B 0,C 180,E1 -6157.562,E2 -6157.562} C_VEL
LIN {X 0,Y 495.773,Z 638.734,A -85,B 0,C 180,E1 -6160.7,E2 -6160.7} C_VEL
LIN {X 0,Y 495.737,Z 638.731,A -85,B 0,C 180,E1 -6164.001,E2 -6164.001} C_VEL
LIN {X 0,Y 495.728,Z 638.74,A -85,B 0,C 180,E1 -6167.117,E2 -6167.117} C_VEL
LIN {X 0,Y 495.761,Z 638.738,A -85,B 0,C 180,E1 -6169.953,E2 -6169.953} C_VEL
LIN {X 0,Y 495.773,Z 638.791,A -85,B 0,C 180,E1 -6170.64,E2 -6170.64} C_VEL
LIN {X 0,Y 497.613,Z 648.052,A -85,B 0,C 180,E1 -6173.113,E2 -6173.113} C_VEL
LIN {X 0,Y 497.875,Z 653.208,A -85,B 0,C 180,E1 -6174.388,E2 -6174.388} C_VEL
LIN {X 0,Y 497.431,Z 666.619,A -85,B 0,C 180,E1 -6177.528,E2 -6177.528} C_VEL
LIN {X 0,Y 497.129,Z 679.138,A -85,B 0,C 180,E1 -6180.343,E2 -6180.343} C_VEL
LIN {X 0,Y 496.822,Z 693.854,A -85,B 0,C 180,E1 -6183.538,E2 -6183.538} C_VEL
LIN {X 0,Y 496.494,Z 708.49,A -85,B 0,C 180,E1 -6186.65,E2 -6186.65} C_VEL
LIN {X 0,Y 496.192,Z 723.302,A -85,B 0,C 180,E1 -6189.695,E2 -6189.695} C_VEL
LIN {X 0,Y 495.968,Z 738.101,A -85,B 0,C 180,E1 -6192.688,E2 -6192.688} C_VEL
LIN {X 0,Y 495.702,Z 751.641,A -85,B 0,C 180,E1 -6195.45,E2 -6195.45} C_VEL
LIN {X 0,Y 497.123,Z 762.88,A -85,B 0,C 180,E1 -6195.728,E2 -6195.728} C_VEL
LIN {X 0,Y 497.72,Z 769.231,A -85,B 0,C 180,E1 -6195.928,E2 -6195.928} C_VEL
LIN {X 0,Y 497.408,Z 781.928,A -85,B 0,C 180,E1 -6196.414,E2 -6196.414} C_VEL
LIN {X 0,Y 497.024,Z 793.524,A -85,B 0,C 180,E1 -6197.01,E2 -6197.01} C_VEL
LIN {X 0,Y 496.671,Z 804.663,A -85,B 0,C 180,E1 -6197.745,E2 -6197.745} C_VEL
LIN {X 0,Y 496.309,Z 815.787,A -85,B 0,C 180,E1 -6198.669,E2 -6198.669} C_VEL
LIN {X 0,Y 495.921,Z 826.694,A -85,B 0,C 180,E1 -6199.796,E2 -6199.796} C_VEL
LIN {X 0,Y 495.637,Z 834.726,A -85,B 0,C 180,E1 -6200.82,E2 -6200.82} C_VEL
LIN {X 0,Y 495.4,Z 842.653,A -85,B 0,C 180,E1 -6202.049,E2 -6202.049} C_VEL
LIN {X 0,Y 495.204,Z 849.927,A -85,B 0,C 180,E1 -6203.48,E2 -6203.48} C_VEL
LIN {X 0,Y 495.123,Z 854.781,A -85,B 0,C 180,E1 -6204.706,E2 -6204.706} C_VEL
LIN {X 0,Y 495.053,Z 858.495,A -85,B 0,C 180,E1 -6205.929,E2 -6205.929} C_VEL
LIN {X 0,Y 495.043,Z 860.417,A -85,B 0,C 180,E1 -6206.744,E2 -6206.744} C_VEL
LIN {X 0,Y 494.974,Z 861.849,A -85,B 0,C 180,E1 -6207.558,E2 -6207.558} C_VEL
LIN {X 0,Y 494.961,Z 862.872,A -85,B 0,C 180,E1 -6208.372,E2 -6208.372} C_VEL
LIN {X 0,Y 494.911,Z 863.491,A -85,B 0,C 180,E1 -6209.186,E2 -6209.186} C_VEL
LIN {X 0,Y 494.898,Z 863.712,A -85,B 0,C 180,E1 -6210,E2 -6210} C_VEL
LIN {X 0,Y 494.911,Z 863.492,A -85,B 0,C 180,E1 -6210.813,E2 -6210.813} C_VEL
LIN {X 0,Y 494.961,Z 862.872,A -85,B 0,C 180,E1 -6211.627,E2 -6211.627} C_VEL
LIN {X 0,Y 494.974,Z 861.849,A -85,B 0,C 180,E1 -6212.441,E2 -6212.441} C_VEL
LIN {X 0,Y 495.043,Z 860.42,A -85,B 0,C 180,E1 -6213.255,E2 -6213.255} C_VEL
LIN {X 0,Y 495.03,Z 857.401,A -85,B 0,C 180,E1 -6214.478,E2 -6214.478} C_VEL
LIN {X 0,Y 495.178,Z 853.332,A -85,B 0,C 180,E1 -6215.701,E2 -6215.701} C_VEL
LIN {X 0,Y 495.251,Z 847.175,A -85,B 0,C 180,E1 -6217.112,E2 -6217.112} C_VEL
LIN {X 0,Y 495.485,Z 840.243,A -85,B 0,C 180,E1 -6218.359,E2 -6218.359} C_VEL
LIN {X 0,Y 495.735,Z 831.795,A -85,B 0,C 180,E1 -6219.588,E2 -6219.588} C_VEL
LIN {X 0,Y 496.012,Z 823.123,A -85,B 0,C 180,E1 -6220.614,E2 -6220.614} C_VEL
LIN {X 0,Y 496.458,Z 812.484,A -85,B 0,C 180,E1 -6221.637,E2 -6221.637} C_VEL
LIN {X 0,Y 496.761,Z 801.012,A -85,B 0,C 180,E1 -6222.528,E2 -6222.528} C_VEL
LIN {X 0,Y 497.109,Z 790.464,A -85,B 0,C 180,E1 -6223.177,E2 -6223.177} C_VEL
LIN {X 0,Y 497.459,Z 778.681,A -85,B 0,C 180,E1 -6223.74,E2 -6223.74} C_VEL
LIN {X 0,Y 497.646,Z 766.514,A -85,B 0,C 180,E1 -6224.164,E2 -6224.164} C_VEL
LIN {X 0,Y 495.838,Z 753.699,A -85,B 0,C 180,E1 -6224.507,E2 -6224.507} C_VEL
LIN {X 0,Y 495.72,Z 751.798,A -85,B 0,C 180,E1 -6224.574,E2 -6224.574} C_VEL
LIN {X 0,Y 495.973,Z 736.394,A -85,B 0,C 180,E1 -6227.737,E2 -6227.737} C_VEL
LIN {X 0,Y 496.3,Z 721.455,A -85,B 0,C 180,E1 -6230.834,E2 -6230.834} C_VEL
LIN {X 0,Y 496.636,Z 706.462,A -85,B 0,C 180,E1 -6234.006,E2 -6234.006} C_VEL
LIN {X 0,Y 497.006,Z 692.589,A -85,B 0,C 180,E1 -6237.018,E2 -6237.018} C_VEL
LIN {X 0,Y 497.406,Z 678.912,A -85,B 0,C 180,E1 -6240.063,E2 -6240.063} C_VEL
LIN {X 0,Y 497.886,Z 665.453,A -85,B 0,C 180,E1 -6243.159,E2 -6243.159} C_VEL
LIN {X 0,Y 498.331,Z 652.197,A -85,B 0,C 180,E1 -6246.322,E2 -6246.322} C_VEL
LIN {X 0,Y 496.793,Z 643.886,A -85,B 0,C 180,E1 -6248.495,E2 -6248.495} C_VEL
LIN {X 0,Y 495.741,Z 638.736,A -85,B 0,C 180,E1 -6249.911,E2 -6249.911} C_VEL
LIN {X 0,Y 495.723,Z 638.739,A -85,B 0,C 180,E1 -6252.882,E2 -6252.882} C_VEL
LIN {X 0,Y 495.734,Z 638.734,A -85,B 0,C 180,E1 -6255.999,E2 -6255.999} C_VEL
LIN {X 0,Y 495.766,Z 638.732,A -85,B 0,C 180,E1 -6258.705,E2 -6258.705} C_VEL
LIN {X 0,Y 495.762,Z 638.728,A -85,B 0,C 180,E1 -6261.409,E2 -6261.409} C_VEL
LIN {X 0,Y 495.753,Z 638.73,A -85,B 0,C 180,E1 -6264.462,E2 -6264.462} C_VEL
LIN {X 0,Y 495.765,Z 638.729,A -85,B 0,C 180,E1 -6267.405,E2 -6267.405} C_VEL
LIN {X 0,Y 495.778,Z 638.727,A -85,B 0,C 180,E1 -6270.254,E2 -6270.254} C_VEL
LIN {X 0,Y 495.829,Z 638.722,A -85,B 0,C 180,E1 -6273.248,E2 -6273.248} C_VEL
LIN {X 0,Y 495.748,Z 638.734,A -85,B 0,C 180,E1 -6275.725,E2 -6275.725} C_VEL
LIN {X 0,Y 495.74,Z 638.731,A -85,B 0,C 180,E1 -6278.371,E2 -6278.371} C_VEL
LIN {X 0,Y 495.78,Z 638.728,A -85,B 0,C 180,E1 -6280.971,E2 -6280.971} C_VEL
LIN {X 0,Y 495.774,Z 638.729,A -85,B 0,C 180,E1 -6283.53,E2 -6283.53} C_VEL
LIN {X 0,Y 495.792,Z 638.724,A -85,B 0,C 180,E1 -6286.055,E2 -6286.055} C_VEL
LIN {X 0,Y 495.87,Z 638.719,A -85,B 0,C 180,E1 -6288.555,E2 -6288.555} C_VEL
LIN {X 0,Y 495.869,Z 638.716,A -85,B 0,C 180,E1 -6291.852,E2 -6291.852} C_VEL
LIN {X 0,Y 495.891,Z 638.718,A -85,B 0,C 180,E1 -6294.306,E2 -6294.306} C_VEL
LIN {X 0,Y 495.988,Z 638.701,A -85,B 0,C 180,E1 -6297.564,E2 -6297.564} C_VEL
LIN {X 0,Y 495.993,Z 638.706,A -85,B 0,C 180,E1 -6300,E2 -6300} C_VEL
LIN {X 0,Y 495.989,Z 638.706,A -85,B 0,C 180,E1 -6302.436,E2 -6302.436} C_VEL
LIN {X 0,Y 495.771,Z 638.771,A -85,B 0,C 180,E1 -6303.912,E2 -6303.912} C_VEL
LIN {X 0,Y 496.59,Z 644.253,A -85,B 0,C 180,E1 -6305.278,E2 -6305.278} C_VEL
LIN {X 0,Y 496.746,Z 657.457,A -85,B 0,C 180,E1 -6308.543,E2 -6308.543} C_VEL
LIN {X 0,Y 496.667,Z 670.505,A -85,B 0,C 180,E1 -6311.84,E2 -6311.84} C_VEL
LIN {X 0,Y 496.46,Z 681.76,A -85,B 0,C 180,E1 -6314.762,E2 -6314.762} C_VEL
LIN {X 0,Y 496.292,Z 693.17,A -85,B 0,C 180,E1 -6317.726,E2 -6317.726} C_VEL
LIN {X 0,Y 496.065,Z 704.679,A -85,B 0,C 180,E1 -6320.765,E2 -6320.765} C_VEL
LIN {X 0,Y 495.819,Z 716.174,A -85,B 0,C 180,E1 -6323.827,E2 -6323.827} C_VEL
LIN {X 0,Y 495.628,Z 726.115,A -85,B 0,C 180,E1 -6326.517,E2 -6326.517} C_VEL
LIN {X 0,Y 497.813,Z 739.839,A -85,B 0,C 180,E1 -6326.913,E2 -6326.913} C_VEL
LIN {X 0,Y 497.523,Z 753.32,A -85,B 0,C 180,E1 -6327.408,E2 -6327.408} C_VEL
LIN {X 0,Y 497.133,Z 765.582,A -85,B 0,C 180,E1 -6328.038,E2 -6328.038} C_VEL
LIN {X 0,Y 496.715,Z 777.891,A -85,B 0,C 180,E1 -6328.871,E2 -6328.871} C_VEL
LIN {X 0,Y 496.384,Z 787.697,A -85,B 0,C 180,E1 -6329.706,E2 -6329.706} C_VEL
LIN {X 0,Y 495.955,Z 797.964,A -85,B 0,C 180,E1 -6330.791,E2 -6330.791} C_VEL
LIN {X 0,Y 495.661,Z 806.399,A -85,B 0,C 180,E1 -6331.892,E2 -6331.892} C_VEL
LIN {X 0,Y 495.413,Z 814.354,A -85,B 0,C 180,E1 -6333.179,E2 -6333.179} C_VEL
LIN {X 0,Y 495.206,Z 821.241,A -85,B 0,C 180,E1 -6334.601,E2 -6334.601} C_VEL
LIN {X 0,Y 495.069,Z 826.383,A -85,B 0,C 180,E1 -6335.986,E2 -6335.986} C_VEL
LIN {X 0,Y 494.984,Z 830.029,A -85,B 0,C 180,E1 -6337.335,E2 -6337.335} C_VEL
LIN {X 0,Y 494.925,Z 832.472,A -85,B 0,C 180,E1 -6338.668,E2 -6338.668} C_VEL
LIN {X 0,Y 494.864,Z 833.788,A -85,B 0,C 180,E1 -6339.925,E2 -6339.925} C_VEL
LIN {X 0,Y 494.851,Z 834.16,A -85,B 0,C 180,E1 -6341.175,E2 -6341.175} C_VEL
LIN {X 0,Y 494.878,Z 833.626,A -85,B 0,C 180,E1 -6342.399,E2 -6342.399} C_VEL
LIN {X 0,Y 494.905,Z 832.232,A -85,B 0,C 180,E1 -6343.596,E2 -6343.596} C_VEL
LIN {X 0,Y 495.016,Z 828.874,A -85,B 0,C 180,E1 -6345.225,E2 -6345.225} C_VEL
LIN {X 0,Y 495.117,Z 824.274,A -85,B 0,C 180,E1 -6346.72,E2 -6346.72} C_VEL
LIN {X 0,Y 495.249,Z 818.485,A -85,B 0,C 180,E1 -6348.099,E2 -6348.099} C_VEL
LIN {X 0,Y 495.493,Z 811.163,A -85,B 0,C 180,E1 -6349.462,E2 -6349.462} C_VEL
LIN {X 0,Y 495.748,Z 803.611,A -85,B 0,C 180,E1 -6350.587,E2 -6350.587} C_VEL
LIN {X 0,Y 495.859,Z 800.575,A -85,B 0,C 180,E1 -6350.979,E2 -6350.979} C_VEL
LIN {X 0,Y 495.354,Z 796.603,A -85,B 0,C 180,E1 -6351.481,E2 -6351.481} C_VEL
LIN {X 0,Y 492.852,Z 789.872,A -85,B 0,C 180,E1 -6352.274,E2 -6352.274} C_VEL
LIN {X 0,Y 490.323,Z 782.622,A -85,B 0,C 180,E1 -6353.005,E2 -6353.005} C_VEL
LIN {X 0,Y 489.774,Z 777.836,A -85,B 0,C 180,E1 -6353.405,E2 -6353.405} C_VEL
LIN {X 0,Y 490.191,Z 766.317,A -85,B 0,C 180,E1 -6354.198,E2 -6354.198} C_VEL
LIN {X 0,Y 490.655,Z 753.741,A -85,B 0,C 180,E1 -6354.86,E2 -6354.86} C_VEL
LIN {X 0,Y 490.857,Z 740.113,A -85,B 0,C 180,E1 -6355.373,E2 -6355.373} C_VEL
LIN {X 0,Y 488.845,Z 727.733,A -85,B 0,C 180,E1 -6355.742,E2 -6355.742} C_VEL
LIN {X 0,Y 488.575,Z 726.206,A -85,B 0,C 180,E1 -6355.782,E2 -6355.782} C_VEL
LIN {X 0,Y 488.815,Z 715.034,A -85,B 0,C 180,E1 -6358.83,E2 -6358.83} C_VEL
LIN {X 0,Y 489.096,Z 704.471,A -85,B 0,C 180,E1 -6361.694,E2 -6361.694} C_VEL
LIN {X 0,Y 489.413,Z 691.977,A -85,B 0,C 180,E1 -6365.09,E2 -6365.09} C_VEL
LIN {X 0,Y 489.633,Z 680.939,A -85,B 0,C 180,E1 -6368.088,E2 -6368.088} C_VEL
LIN {X 0,Y 489.859,Z 671.18,A -85,B 0,C 180,E1 -6370.733,E2 -6370.733} C_VEL
LIN {X 0,Y 490.016,Z 659.349,A -85,B 0,C 180,E1 -6373.933,E2 -6373.933} C_VEL
LIN {X 0,Y 490.083,Z 648.975,A -85,B 0,C 180,E1 -6376.736,E2 -6376.736} C_VEL
LIN {X 0,Y 489.421,Z 642.96,A -85,B 0,C 180,E1 -6378.403,E2 -6378.403} C_VEL
LIN {X 0,Y 488.76,Z 639.604,A -85,B 0,C 180,E1 -6379.384,E2 -6379.384} C_VEL
LIN {X 0,Y 488.873,Z 639.593,A -85,B 0,C 180,E1 -6382.719,E2 -6382.719} C_VEL
LIN {X 0,Y 488.814,Z 639.6,A -85,B 0,C 180,E1 -6385.052,E2 -6385.052} C_VEL
LIN {X 0,Y 488.963,Z 639.58,A -85,B 0,C 180,E1 -6387.529,E2 -6387.529} C_VEL
LIN {X 0,Y 488.957,Z 639.581,A -85,B 0,C 180,E1 -6390.824,E2 -6390.824} C_VEL
LIN {X 0,Y 488.963,Z 639.579,A -85,B 0,C 180,E1 -6392.472,E2 -6392.472} C_VEL
LIN {X 0,Y 488.849,Z 639.594,A -85,B 0,C 180,E1 -6395.776,E2 -6395.776} C_VEL
LIN {X 0,Y 488.82,Z 639.597,A -85,B 0,C 180,E1 -6398.267,E2 -6398.267} C_VEL
LIN {X 0,Y 488.832,Z 639.596,A -85,B 0,C 180,E1 -6401.612,E2 -6401.612} C_VEL
LIN {X 0,Y 488.765,Z 639.604,A -85,B 0,C 180,E1 -6405.001,E2 -6405.001} C_VEL
LIN {X 0,Y 488.757,Z 639.605,A -85,B 0,C 180,E1 -6408.442,E2 -6408.442} C_VEL
LIN {X 0,Y 488.709,Z 639.612,A -85,B 0,C 180,E1 -6411.071,E2 -6411.071} C_VEL
LIN {X 0,Y 488.754,Z 639.606,A -85,B 0,C 180,E1 -6414.081,E2 -6414.081} C_VEL
LIN {X 0,Y 490.853,Z 647.259,A -85,B 0,C 180,E1 -6414.533,E2 -6414.533} C_VEL
LIN {X 0,Y 490.698,Z 658.628,A -85,B 0,C 180,E1 -6415.22,E2 -6415.22} C_VEL
LIN {X 0,Y 490.306,Z 669.427,A -85,B 0,C 180,E1 -6416.038,E2 -6416.038} C_VEL
LIN {X 0,Y 489.989,Z 679.261,A -85,B 0,C 180,E1 -6416.973,E2 -6416.973} C_VEL
LIN {X 0,Y 489.629,Z 688.411,A -85,B 0,C 180,E1 -6418.04,E2 -6418.04} C_VEL
LIN {X 0,Y 489.279,Z 696.743,A -85,B 0,C 180,E1 -6419.234,E2 -6419.234} C_VEL
LIN {X 0,Y 489.026,Z 703.465,A -85,B 0,C 180,E1 -6420.426,E2 -6420.426} C_VEL
LIN {X 0,Y 488.802,Z 708.684,A -85,B 0,C 180,E1 -6421.568,E2 -6421.568} C_VEL
LIN {X 0,Y 488.675,Z 712.619,A -85,B 0,C 180,E1 -6422.637,E2 -6422.637} C_VEL
LIN {X 0,Y 488.506,Z 716.834,A -85,B 0,C 180,E1 -6424.131,E2 -6424.131} C_VEL
LIN {X 0,Y 488.42,Z 718.84,A -85,B 0,C 180,E1 -6425.14,E2 -6425.14} C_VEL
LIN {X 0,Y 488.352,Z 720.424,A -85,B 0,C 180,E1 -6426.302,E2 -6426.302} C_VEL
LIN {X 0,Y 488.324,Z 721.288,A -85,B 0,C 180,E1 -6427.668,E2 -6427.668} C_VEL
LIN {X 0,Y 488.376,Z 720.956,A -85,B 0,C 180,E1 -6429.286,E2 -6429.286} C_VEL
LIN {X 0,Y 488.427,Z 719.889,A -85,B 0,C 180,E1 -6430.354,E2 -6430.354} C_VEL
LIN {X 0,Y 488.564,Z 716.953,A -85,B 0,C 180,E1 -6432.011,E2 -6432.011} C_VEL
LIN {X 0,Y 488.694,Z 713.793,A -85,B 0,C 180,E1 -6433.192,E2 -6433.192} C_VEL
LIN {X 0,Y 488.828,Z 709.696,A -85,B 0,C 180,E1 -6434.367,E2 -6434.367} C_VEL
LIN {X 0,Y 489.067,Z 704.584,A -85,B 0,C 180,E1 -6435.533,E2 -6435.533} C_VEL
LIN {X 0,Y 489.308,Z 698.256,A -85,B 0,C 180,E1 -6436.703,E2 -6436.703} C_VEL
LIN {X 0,Y 489.681,Z 689.733,A -85,B 0,C 180,E1 -6437.964,E2 -6437.964} C_VEL
LIN {X 0,Y 490.068,Z 679.956,A -85,B 0,C 180,E1 -6439.124,E2 -6439.124} C_VEL
LIN {X 0,Y 490.447,Z 670.032,A -85,B 0,C 180,E1 -6440.069,E2 -6440.069} C_VEL
LIN {X 0,Y 490.79,Z 658.447,A -85,B 0,C 180,E1 -6440.945,E2 -6440.945} C_VEL
LIN {X 0,Y 490.914,Z 647.219,A -85,B 0,C 180,E1 -6441.614,E2 -6441.614} C_VEL
LIN {X 0,Y 488.701,Z 639.612,A -85,B 0,C 180,E1 -6442.065,E2 -6442.065} C_VEL
LIN {X 0,Y 488.724,Z 639.607,A -85,B 0,C 180,E1 -6445.053,E2 -6445.053} C_VEL
LIN {X 0,Y 488.704,Z 639.61,A -85,B 0,C 180,E1 -6448.046,E2 -6448.046} C_VEL
LIN {X 0,Y 488.724,Z 639.603,A -85,B 0,C 180,E1 -6450.73,E2 -6450.73} C_VEL
LIN {X 0,Y 488.754,Z 639.604,A -85,B 0,C 180,E1 -6453.528,E2 -6453.528} C_VEL
LIN {X 0,Y 488.677,Z 639.608,A -85,B 0,C 180,E1 -6456.254,E2 -6456.254} C_VEL
LIN {X 0,Y 488.747,Z 639.603,A -85,B 0,C 180,E1 -6459.176,E2 -6459.176} C_VEL
LIN {X 0,Y 488.735,Z 639.603,A -85,B 0,C 180,E1 -6462.424,E2 -6462.424} C_VEL
LIN {X 0,Y 488.763,Z 639.599,A -85,B 0,C 180,E1 -6465,E2 -6465} C_VEL
LIN {X 0,Y 488.806,Z 639.593,A -85,B 0,C 180,E1 -6468.388,E2 -6468.388} C_VEL
LIN {X 0,Y 488.819,Z 639.597,A -85,B 0,C 180,E1 -6471.734,E2 -6471.734} C_VEL
LIN {X 0,Y 488.856,Z 639.592,A -85,B 0,C 180,E1 -6474.224,E2 -6474.224} C_VEL
LIN {X 0,Y 488.963,Z 639.572,A -85,B 0,C 180,E1 -6477.529,E2 -6477.529} C_VEL
LIN {X 0,Y 488.956,Z 639.57,A -85,B 0,C 180,E1 -6480.824,E2 -6480.824} C_VEL
LIN {X 0,Y 488.963,Z 639.576,A -85,B 0,C 180,E1 -6482.471,E2 -6482.471} C_VEL
LIN {X 0,Y 488.856,Z 639.586,A -85,B 0,C 180,E1 -6485.776,E2 -6485.776} C_VEL
LIN {X 0,Y 488.819,Z 639.595,A -85,B 0,C 180,E1 -6488.266,E2 -6488.266} C_VEL
LIN {X 0,Y 488.807,Z 639.594,A -85,B 0,C 180,E1 -6491.613,E2 -6491.613} C_VEL
LIN {X 0,Y 488.763,Z 639.599,A -85,B 0,C 180,E1 -6495,E2 -6495} C_VEL
LIN {X 0,Y 488.757,Z 639.605,A -85,B 0,C 180,E1 -6498.442,E2 -6498.442} C_VEL
LIN {X 0,Y 488.708,Z 639.606,A -85,B 0,C 180,E1 -6501.071,E2 -6501.071} C_VEL
LIN {X 0,Y 488.691,Z 639.607,A -85,B 0,C 180,E1 -6503.746,E2 -6503.746} C_VEL
LIN {X 0,Y 488.794,Z 639.597,A -85,B 0,C 180,E1 -6506.944,E2 -6506.944} C_VEL
LIN {X 0,Y 488.712,Z 639.612,A -85,B 0,C 180,E1 -6510.363,E2 -6510.363} C_VEL
LIN {X 0,Y 488.736,Z 639.603,A -85,B 0,C 180,E1 -6513.484,E2 -6513.484} C_VEL
LIN {X 0,Y 488.684,Z 639.616,A -85,B 0,C 180,E1 -6516.355,E2 -6516.355} C_VEL
LIN {X 0,Y 488.704,Z 639.609,A -85,B 0,C 180,E1 -6519.254,E2 -6519.254} C_VEL
LIN {X 0,Y 488.713,Z 639.606,A -85,B 0,C 180,E1 -6521.6,E2 -6521.6} C_VEL
LIN {X 0,Y 488.715,Z 639.612,A -85,B 0,C 180,E1 -6524.801,E2 -6524.801} C_VEL
LIN {X 0,Y 488.694,Z 639.614,A -85,B 0,C 180,E1 -6527.475,E2 -6527.475} C_VEL
LIN {X 0,Y 488.747,Z 639.813,A -85,B 0,C 180,E1 -6530.417,E2 -6530.417} C_VEL
LIN {X 0,Y 490.643,Z 649.387,A -85,B 0,C 180,E1 -6533.014,E2 -6533.014} C_VEL
LIN {X 0,Y 490.968,Z 653.51,A -85,B 0,C 180,E1 -6534.063,E2 -6534.063} C_VEL
LIN {X 0,Y 490.526,Z 665.818,A -85,B 0,C 180,E1 -6537.013,E2 -6537.013} C_VEL
LIN {X 0,Y 490.154,Z 678.257,A -85,B 0,C 180,E1 -6539.878,E2 -6539.878} C_VEL
LIN {X 0,Y 489.84,Z 691.453,A -85,B 0,C 180,E1 -6542.817,E2 -6542.817} C_VEL
LIN {X 0,Y 489.501,Z 705.469,A -85,B 0,C 180,E1 -6545.846,E2 -6545.846} C_VEL
LIN {X 0,Y 489.177,Z 720.606,A -85,B 0,C 180,E1 -6549.044,E2 -6549.044} C_VEL
LIN {X 0,Y 488.893,Z 736.976,A -85,B 0,C 180,E1 -6552.429,E2 -6552.429} C_VEL
LIN {X 0,Y 488.628,Z 750.512,A -85,B 0,C 180,E1 -6555.235,E2 -6555.235} C_VEL
LIN {X 0,Y 489.873,Z 761.542,A -85,B 0,C 180,E1 -6555.508,E2 -6555.508} C_VEL
LIN {X 0,Y 490.757,Z 769.629,A -85,B 0,C 180,E1 -6555.777,E2 -6555.777} C_VEL
LIN {X 0,Y 490.424,Z 781.933,A -85,B 0,C 180,E1 -6556.27,E2 -6556.27} C_VEL
LIN {X 0,Y 489.982,Z 794.255,A -85,B 0,C 180,E1 -6556.933,E2 -6556.933} C_VEL
LIN {X 0,Y 489.574,Z 806.22,A -85,B 0,C 180,E1 -6557.775,E2 -6557.775} C_VEL
LIN {X 0,Y 489.232,Z 816.871,A -85,B 0,C 180,E1 -6558.712,E2 -6558.712} C_VEL
LIN {X 0,Y 488.847,Z 825.574,A -85,B 0,C 180,E1 -6559.647,E2 -6559.647} C_VEL
LIN {X 0,Y 488.57,Z 833.61,A -85,B 0,C 180,E1 -6560.687,E2 -6560.687} C_VEL
LIN {X 0,Y 488.35,Z 841.586,A -85,B 0,C 180,E1 -6561.934,E2 -6561.934} C_VEL
LIN {X 0,Y 488.142,Z 849.034,A -85,B 0,C 180,E1 -6563.428,E2 -6563.428} C_VEL
LIN {X 0,Y 488.089,Z 853.71,A -85,B 0,C 180,E1 -6564.629,E2 -6564.629} C_VEL
LIN {X 0,Y 488.012,Z 857.432,A -85,B 0,C 180,E1 -6565.87,E2 -6565.87} C_VEL
LIN {X 0,Y 487.999,Z 859.363,A -85,B 0,C 180,E1 -6566.697,E2 -6566.697} C_VEL
LIN {X 0,Y 487.938,Z 860.834,A -85,B 0,C 180,E1 -6567.523,E2 -6567.523} C_VEL
LIN {X 0,Y 487.929,Z 861.843,A -85,B 0,C 180,E1 -6568.349,E2 -6568.349} C_VEL
LIN {X 0,Y 487.884,Z 862.468,A -85,B 0,C 180,E1 -6569.174,E2 -6569.174} C_VEL
LIN {X 0,Y 487.871,Z 862.698,A -85,B 0,C 180,E1 -6570,E2 -6570} C_VEL
LIN {X 0,Y 487.881,Z 862.489,A -85,B 0,C 180,E1 -6570.825,E2 -6570.825} C_VEL
LIN {X 0,Y 487.936,Z 860.847,A -85,B 0,C 180,E1 -6572.476,E2 -6572.476} C_VEL
LIN {X 0,Y 487.999,Z 859.415,A -85,B 0,C 180,E1 -6573.302,E2 -6573.302} C_VEL
LIN {X 0,Y 487.983,Z 856.382,A -85,B 0,C 180,E1 -6574.543,E2 -6574.543} C_VEL
LIN {X 0,Y 488.127,Z 852.302,A -85,B 0,C 180,E1 -6575.784,E2 -6575.784} C_VEL
LIN {X 0,Y 488.183,Z 846.074,A -85,B 0,C 180,E1 -6577.236,E2 -6577.236} C_VEL
LIN {X 0,Y 488.441,Z 839.23,A -85,B 0,C 180,E1 -6578.481,E2 -6578.481} C_VEL
LIN {X 0,Y 488.685,Z 830.789,A -85,B 0,C 180,E1 -6579.728,E2 -6579.728} C_VEL
LIN {X 0,Y 488.97,Z 822.097,A -85,B 0,C 180,E1 -6580.768,E2 -6580.768} C_VEL
LIN {X 0,Y 489.428,Z 811.467,A -85,B 0,C 180,E1 -6581.807,E2 -6581.807} C_VEL
LIN {X 0,Y 489.79,Z 799.699,A -85,B 0,C 180,E1 -6582.731,E2 -6582.731} C_VEL
LIN {X 0,Y 490.222,Z 787.498,A -85,B 0,C 180,E1 -6583.471,E2 -6583.471} C_VEL
LIN {X 0,Y 490.551,Z 775.047,A -85,B 0,C 180,E1 -6584.043,E2 -6584.043} C_VEL
LIN {X 0,Y 490.658,Z 766.88,A -85,B 0,C 180,E1 -6584.331,E2 -6584.331} C_VEL
LIN {X 0,Y 489.016,Z 755.059,A -85,B 0,C 180,E1 -6584.672,E2 -6584.672} C_VEL
LIN {X 0,Y 488.613,Z 750.807,A -85,B 0,C 180,E1 -6584.791,E2 -6584.791} C_VEL
LIN {X 0,Y 488.899,Z 736.468,A -85,B 0,C 180,E1 -6587.786,E2 -6587.786} C_VEL
LIN {X 0,Y 489.244,Z 721.089,A -85,B 0,C 180,E1 -6591.046,E2 -6591.046} C_VEL
LIN {X 0,Y 489.64,Z 705.69,A -85,B 0,C 180,E1 -6594.371,E2 -6594.371} C_VEL
LIN {X 0,Y 490.01,Z 692.365,A -85,B 0,C 180,E1 -6597.319,E2 -6597.319} C_VEL
LIN {X 0,Y 490.473,Z 678.742,A -85,B 0,C 180,E1 -6600.413,E2 -6600.413} C_VEL
LIN {X 0,Y 491.03,Z 663.924,A -85,B 0,C 180,E1 -6603.886,E2 -6603.886} C_VEL
LIN {X 0,Y 491.419,Z 653.94,A -85,B 0,C 180,E1 -6606.317,E2 -6606.317} C_VEL
LIN {X 0,Y 490.072,Z 646.332,A -85,B 0,C 180,E1 -6608.328,E2 -6608.328} C_VEL
LIN {X 0,Y 488.708,Z 639.612,A -85,B 0,C 180,E1 -6610.19,E2 -6610.19} C_VEL
LIN {X 0,Y 488.707,Z 639.613,A -85,B 0,C 180,E1 -6612.826,E2 -6612.826} C_VEL
LIN {X 0,Y 488.7,Z 639.61,A -85,B 0,C 180,E1 -6615.975,E2 -6615.975} C_VEL
LIN {X 0,Y 488.721,Z 639.611,A -85,B 0,C 180,E1 -6618.585,E2 -6618.585} C_VEL
LIN {X 0,Y 488.746,Z 639.603,A -85,B 0,C 180,E1 -6620.94,E2 -6620.94} C_VEL
LIN {X 0,Y 488.681,Z 639.613,A -85,B 0,C 180,E1 -6623.868,E2 -6623.868} C_VEL
LIN {X 0,Y 488.735,Z 639.603,A -85,B 0,C 180,E1 -6626.877,E2 -6626.877} C_VEL
LIN {X 0,Y 488.73,Z 639.609,A -85,B 0,C 180,E1 -6629.781,E2 -6629.781} C_VEL
LIN {X 0,Y 488.795,Z 639.597,A -85,B 0,C 180,E1 -6633.054,E2 -6633.054} C_VEL
LIN {X 0,Y 488.689,Z 639.609,A -85,B 0,C 180,E1 -6636.254,E2 -6636.254} C_VEL
LIN {X 0,Y 488.741,Z 639.608,A -85,B 0,C 180,E1 -6639.175,E2 -6639.175} C_VEL
LIN {X 0,Y 488.754,Z 639.602,A -85,B 0,C 180,E1 -6641.627,E2 -6641.627} C_VEL
LIN {X 0,Y 488.757,Z 639.604,A -85,B 0,C 180,E1 -6644.999,E2 -6644.999} C_VEL
LIN {X 0,Y 488.828,Z 639.594,A -85,B 0,C 180,E1 -6648.388,E2 -6648.388} C_VEL
LIN {X 0,Y 488.813,Z 639.594,A -85,B 0,C 180,E1 -6651.733,E2 -6651.733} C_VEL
LIN {X 0,Y 488.85,Z 639.594,A -85,B 0,C 180,E1 -6654.224,E2 -6654.224} C_VEL
LIN {X 0,Y 488.956,Z 639.577,A -85,B 0,C 180,E1 -6657.528,E2 -6657.528} C_VEL
LIN {X 0,Y 488.949,Z 639.581,A -85,B 0,C 180,E1 -6660.823,E2 -6660.823} C_VEL
LIN {X 0,Y 488.957,Z 639.582,A -85,B 0,C 180,E1 -6662.471,E2 -6662.471} C_VEL
LIN {X 0,Y 488.775,Z 639.777,A -85,B 0,C 180,E1 -6663.761,E2 -6663.761} C_VEL
LIN {X 0,Y 489.64,Z 646.064,A -85,B 0,C 180,E1 -6665.353,E2 -6665.353} C_VEL
LIN {X 0,Y 489.772,Z 657.692,A -85,B 0,C 180,E1 -6668.25,E2 -6668.25} C_VEL
LIN {X 0,Y 489.647,Z 669.239,A -85,B 0,C 180,E1 -6671.173,E2 -6671.173} C_VEL
LIN {X 0,Y 489.549,Z 679.012,A -85,B 0,C 180,E1 -6673.702,E2 -6673.702} C_VEL
LIN {X 0,Y 489.29,Z 690.293,A -85,B 0,C 180,E1 -6676.695,E2 -6676.695} C_VEL
LIN {X 0,Y 489.134,Z 700.187,A -85,B 0,C 180,E1 -6679.297,E2 -6679.297} C_VEL
LIN {X 0,Y 488.935,Z 710.16,A -85,B 0,C 180,E1 -6681.946,E2 -6681.946} C_VEL
LIN {X 0,Y 488.694,Z 721.667,A -85,B 0,C 180,E1 -6685.042,E2 -6685.042} C_VEL
LIN {X 0,Y 488.597,Z 726.351,A -85,B 0,C 180,E1 -6686.309,E2 -6686.309} C_VEL
LIN {X 0,Y 490.914,Z 740.315,A -85,B 0,C 180,E1 -6686.723,E2 -6686.723} C_VEL
LIN {X 0,Y 490.647,Z 752.846,A -85,B 0,C 180,E1 -6687.189,E2 -6687.189} C_VEL
LIN {X 0,Y 490.234,Z 764.662,A -85,B 0,C 180,E1 -6687.787,E2 -6687.787} C_VEL
LIN {X 0,Y 489.832,Z 776.295,A -85,B 0,C 180,E1 -6688.564,E2 -6688.564} C_VEL
LIN {X 0,Y 489.412,Z 786.978,A -85,B 0,C 180,E1 -6689.461,E2 -6689.461} C_VEL
LIN {X 0,Y 489.021,Z 796.315,A -85,B 0,C 180,E1 -6690.426,E2 -6690.426} C_VEL
LIN {X 0,Y 488.757,Z 804.177,A -85,B 0,C 180,E1 -6691.416,E2 -6691.416} C_VEL
LIN {X 0,Y 488.443,Z 812.214,A -85,B 0,C 180,E1 -6692.654,E2 -6692.654} C_VEL
LIN {X 0,Y 488.264,Z 818.025,A -85,B 0,C 180,E1 -6693.75,E2 -6693.75} C_VEL
LIN {X 0,Y 488.06,Z 824.034,A -85,B 0,C 180,E1 -6695.169,E2 -6695.169} C_VEL
LIN {X 0,Y 487.916,Z 828.841,A -85,B 0,C 180,E1 -6696.71,E2 -6696.71} C_VEL
LIN {X 0,Y 487.844,Z 832.137,A -85,B 0,C 180,E1 -6698.277,E2 -6698.277} C_VEL
LIN {X 0,Y 487.798,Z 833.515,A -85,B 0,C 180,E1 -6699.341,E2 -6699.341} C_VEL
LIN {X 0,Y 487.755,Z 834.265,A -85,B 0,C 180,E1 -6700.421,E2 -6700.421} C_VEL
LIN {X 0,Y 487.767,Z 834.293,A -85,B 0,C 180,E1 -6701.513,E2 -6701.513} C_VEL
LIN {X 0,Y 487.781,Z 833.547,A -85,B 0,C 180,E1 -6702.71,E2 -6702.71} C_VEL
LIN {X 0,Y 487.853,Z 831.939,A -85,B 0,C 180,E1 -6703.922,E2 -6703.922} C_VEL
LIN {X 0,Y 487.922,Z 829.51,A -85,B 0,C 180,E1 -6705.107,E2 -6705.107} C_VEL
LIN {X 0,Y 488.005,Z 826.252,A -85,B 0,C 180,E1 -6706.27,E2 -6706.27} C_VEL
LIN {X 0,Y 488.17,Z 820.917,A -85,B 0,C 180,E1 -6707.696,E2 -6707.696} C_VEL
LIN {X 0,Y 488.367,Z 814.124,A -85,B 0,C 180,E1 -6709.098,E2 -6709.098} C_VEL
LIN {X 0,Y 488.611,Z 807.286,A -85,B 0,C 180,E1 -6710.223,E2 -6710.223} C_VEL
LIN {X 0,Y 488.955,Z 798.193,A -85,B 0,C 180,E1 -6711.432,E2 -6711.432} C_VEL
LIN {X 0,Y 489.38,Z 788.008,A -85,B 0,C 180,E1 -6712.528,E2 -6712.528} C_VEL
LIN {X 0,Y 489.774,Z 777.836,A -85,B 0,C 180,E1 -6713.405,E2 -6713.405} C_VEL
LIN {X 0,Y 489.256,Z 772.951,A -85,B 0,C 180,E1 -6713.785,E2 -6713.785} C_VEL
LIN {X 0,Y 486.798,Z 764.78,A -85,B 0,C 180,E1 -6714.391,E2 -6714.391} C_VEL
LIN {X 0,Y 484.312,Z 756.341,A -85,B 0,C 180,E1 -6714.923,E2 -6714.923} C_VEL
LIN {X 0,Y 483.802,Z 750.922,A -85,B 0,C 180,E1 -6715.188,E2 -6715.188} C_VEL
LIN {X 0,Y 483.953,Z 740.642,A -85,B 0,C 180,E1 -6715.567,E2 -6715.567} C_VEL
LIN {X 0,Y 481.72,Z 727.566,A -85,B 0,C 180,E1 -6715.967,E2 -6715.967} C_VEL
LIN {X 0,Y 481.546,Z 726.309,A -85,B 0,C 180,E1 -6716.023,E2 -6716.023} C_VEL
LIN {X 0,Y 481.831,Z 714.293,A -85,B 0,C 180,E1 -6719.303,E2 -6719.303} C_VEL
LIN {X 0,Y 482.111,Z 703.75,A -85,B 0,C 180,E1 -6722.195,E2 -6722.195} C_VEL
LIN {X 0,Y 482.388,Z 693.489,A -85,B 0,C 180,E1 -6725.008,E2 -6725.008} C_VEL
LIN {X 0,Y 482.663,Z 681.799,A -85,B 0,C 180,E1 -6728.205,E2 -6728.205} C_VEL
LIN {X 0,Y 482.911,Z 670.369,A -85,B 0,C 180,E1 -6731.327,E2 -6731.327} C_VEL
LIN {X 0,Y 483.087,Z 659.154,A -85,B 0,C 180,E1 -6734.387,E2 -6734.387} C_VEL
LIN {X 0,Y 483.131,Z 650.221,A -85,B 0,C 180,E1 -6736.822,E2 -6736.822} C_VEL
LIN {X 0,Y 482.365,Z 643.678,A -85,B 0,C 180,E1 -6738.657,E2 -6738.657} C_VEL
LIN {X 0,Y 481.727,Z 640.482,A -85,B 0,C 180,E1 -6739.599,E2 -6739.599} C_VEL
LIN {X 0,Y 481.826,Z 640.471,A -85,B 0,C 180,E1 -6742.684,E2 -6742.684} C_VEL
LIN {X 0,Y 481.784,Z 640.475,A -85,B 0,C 180,E1 -6744.979,E2 -6744.979} C_VEL
LIN {X 0,Y 481.93,Z 640.456,A -85,B 0,C 180,E1 -6747.493,E2 -6747.493} C_VEL
LIN {X 0,Y 481.908,Z 640.459,A -85,B 0,C 180,E1 -6750.836,E2 -6750.836} C_VEL
LIN {X 0,Y 481.93,Z 640.455,A -85,B 0,C 180,E1 -6752.508,E2 -6752.508} C_VEL
LIN {X 0,Y 481.809,Z 640.471,A -85,B 0,C 180,E1 -6755.861,E2 -6755.861} C_VEL
LIN {X 0,Y 481.765,Z 640.476,A -85,B 0,C 180,E1 -6758.389,E2 -6758.389} C_VEL
LIN {X 0,Y 481.797,Z 640.471,A -85,B 0,C 180,E1 -6761.784,E2 -6761.784} C_VEL
LIN {X 0,Y 481.745,Z 640.48,A -85,B 0,C 180,E1 -6765.224,E2 -6765.224} C_VEL
LIN {X 0,Y 481.714,Z 640.482,A -85,B 0,C 180,E1 -6768.722,E2 -6768.722} C_VEL
LIN {X 0,Y 481.647,Z 640.491,A -85,B 0,C 180,E1 -6771.395,E2 -6771.395} C_VEL
LIN {X 0,Y 481.706,Z 640.627,A -85,B 0,C 180,E1 -6773.883,E2 -6773.883} C_VEL
LIN {X 0,Y 483.865,Z 648.257,A -85,B 0,C 180,E1 -6774.34,E2 -6774.34} C_VEL
LIN {X 0,Y 484.021,Z 653.931,A -85,B 0,C 180,E1 -6774.674,E2 -6774.674} C_VEL
LIN {X 0,Y 483.688,Z 665.384,A -85,B 0,C 180,E1 -6775.462,E2 -6775.462} C_VEL
LIN {X 0,Y 483.261,Z 675.456,A -85,B 0,C 180,E1 -6776.331,E2 -6776.331} C_VEL
LIN {X 0,Y 482.9,Z 685.429,A -85,B 0,C 180,E1 -6777.405,E2 -6777.405} C_VEL
LIN {X 0,Y 482.524,Z 693.678,A -85,B 0,C 180,E1 -6778.49,E2 -6778.49} C_VEL
LIN {X 0,Y 482.191,Z 701.225,A -85,B 0,C 180,E1 -6779.707,E2 -6779.707} C_VEL
LIN {X 0,Y 481.96,Z 707.352,A -85,B 0,C 180,E1 -6780.932,E2 -6780.932} C_VEL
LIN {X 0,Y 481.737,Z 712.42,A -85,B 0,C 180,E1 -6782.204,E2 -6782.204} C_VEL
LIN {X 0,Y 481.555,Z 716.926,A -85,B 0,C 180,E1 -6783.708,E2 -6783.708} C_VEL
LIN {X 0,Y 481.395,Z 719.954,A -85,B 0,C 180,E1 -6785.159,E2 -6785.159} C_VEL
LIN {X 0,Y 481.315,Z 721.889,A -85,B 0,C 180,E1 -6786.775,E2 -6786.775} C_VEL
LIN {X 0,Y 481.332,Z 722.371,A -85,B 0,C 180,E1 -6787.958,E2 -6787.958} C_VEL
LIN {X 0,Y 481.364,Z 721.983,A -85,B 0,C 180,E1 -6789.303,E2 -6789.303} C_VEL
LIN {X 0,Y 481.426,Z 720.635,A -85,B 0,C 180,E1 -6790.614,E2 -6790.614} C_VEL
LIN {X 0,Y 481.567,Z 717.749,A -85,B 0,C 180,E1 -6792.17,E2 -6792.17} C_VEL
LIN {X 0,Y 481.71,Z 714.761,A -85,B 0,C 180,E1 -6793.292,E2 -6793.292} C_VEL
LIN {X 0,Y 481.9,Z 709.688,A -85,B 0,C 180,E1 -6794.723,E2 -6794.723} C_VEL
LIN {X 0,Y 482.232,Z 702.962,A -85,B 0,C 180,E1 -6796.17,E2 -6796.17} C_VEL
LIN {X 0,Y 482.577,Z 695.898,A -85,B 0,C 180,E1 -6797.375,E2 -6797.375} C_VEL
LIN {X 0,Y 482.897,Z 687.513,A -85,B 0,C 180,E1 -6798.532,E2 -6798.532} C_VEL
LIN {X 0,Y 483.321,Z 678.409,A -85,B 0,C 180,E1 -6799.552,E2 -6799.552} C_VEL
LIN {X 0,Y 483.694,Z 668.381,A -85,B 0,C 180,E1 -6800.467,E2 -6800.467} C_VEL
LIN {X 0,Y 484.034,Z 656.971,A -85,B 0,C 180,E1 -6801.299,E2 -6801.299} C_VEL
LIN {X 0,Y 484.25,Z 649.415,A -85,B 0,C 180,E1 -6801.74,E2 -6801.74} C_VEL
LIN {X 0,Y 481.658,Z 640.488,A -85,B 0,C 180,E1 -6802.288,E2 -6802.288} C_VEL
LIN {X 0,Y 481.689,Z 640.485,A -85,B 0,C 180,E1 -6805.318,E2 -6805.318} C_VEL
LIN {X 0,Y 481.645,Z 640.488,A -85,B 0,C 180,E1 -6808.312,E2 -6808.312} C_VEL
LIN {X 0,Y 481.701,Z 640.481,A -85,B 0,C 180,E1 -6811.219,E2 -6811.219} C_VEL
LIN {X 0,Y 481.69,Z 640.484,A -85,B 0,C 180,E1 -6814.042,E2 -6814.042} C_VEL
LIN {X 0,Y 481.675,Z 640.478,A -85,B 0,C 180,E1 -6816.812,E2 -6816.812} C_VEL
LIN {X 0,Y 481.696,Z 640.485,A -85,B 0,C 180,E1 -6819.503,E2 -6819.503} C_VEL
LIN {X 0,Y 481.708,Z 640.481,A -85,B 0,C 180,E1 -6822.159,E2 -6822.159} C_VEL
LIN {X 0,Y 481.744,Z 640.474,A -85,B 0,C 180,E1 -6824.776,E2 -6824.776} C_VEL
LIN {X 0,Y 481.752,Z 640.474,A -85,B 0,C 180,E1 -6828.215,E2 -6828.215} C_VEL
LIN {X 0,Y 481.764,Z 640.474,A -85,B 0,C 180,E1 -6831.612,E2 -6831.612} C_VEL
LIN {X 0,Y 481.817,Z 640.47,A -85,B 0,C 180,E1 -6834.14,E2 -6834.14} C_VEL
LIN {X 0,Y 481.93,Z 640.447,A -85,B 0,C 180,E1 -6837.493,E2 -6837.493} C_VEL
LIN {X 0,Y 481.907,Z 640.448,A -85,B 0,C 180,E1 -6840.836,E2 -6840.836} C_VEL
LIN {X 0,Y 481.93,Z 640.452,A -85,B 0,C 180,E1 -6842.508,E2 -6842.508} C_VEL
LIN {X 0,Y 481.817,Z 640.464,A -85,B 0,C 180,E1 -6845.861,E2 -6845.861} C_VEL
LIN {X 0,Y 481.764,Z 640.472,A -85,B 0,C 180,E1 -6848.388,E2 -6848.388} C_VEL
LIN {X 0,Y 481.752,Z 640.474,A -85,B 0,C 180,E1 -6851.785,E2 -6851.785} C_VEL
LIN {X 0,Y 481.744,Z 640.472,A -85,B 0,C 180,E1 -6855.224,E2 -6855.224} C_VEL
LIN {X 0,Y 481.713,Z 640.479,A -85,B 0,C 180,E1 -6858.722,E2 -6858.722} C_VEL
LIN {X 0,Y 481.647,Z 640.485,A -85,B 0,C 180,E1 -6861.395,E2 -6861.395} C_VEL
LIN {X 0,Y 481.676,Z 640.484,A -85,B 0,C 180,E1 -6864.113,E2 -6864.113} C_VEL
LIN {X 0,Y 481.749,Z 640.473,A -85,B 0,C 180,E1 -6867.139,E2 -6867.139} C_VEL
LIN {X 0,Y 481.681,Z 640.482,A -85,B 0,C 180,E1 -6869.741,E2 -6869.741} C_VEL
LIN {X 0,Y 481.674,Z 640.488,A -85,B 0,C 180,E1 -6872.674,E2 -6872.674} C_VEL
LIN {X 0,Y 481.638,Z 640.488,A -85,B 0,C 180,E1 -6875.71,E2 -6875.71} C_VEL
LIN {X 0,Y 481.674,Z 640.489,A -85,B 0,C 180,E1 -6878.859,E2 -6878.859} C_VEL
LIN {X 0,Y 481.657,Z 640.486,A -85,B 0,C 180,E1 -6881.913,E2 -6881.913} C_VEL
LIN {X 0,Y 481.662,Z 640.489,A -85,B 0,C 180,E1 -6884.457,E2 -6884.457} C_VEL
LIN {X 0,Y 481.65,Z 640.491,A -85,B 0,C 180,E1 -6887.839,E2 -6887.839} C_VEL
LIN {X 0,Y 481.723,Z 640.563,A -85,B 0,C 180,E1 -6890.103,E2 -6890.103} C_VEL
LIN {X 0,Y 483.762,Z 651.13,A -85,B 0,C 180,E1 -6893.038,E2 -6893.038} C_VEL
LIN {X 0,Y 484.025,Z 654.811,A -85,B 0,C 180,E1 -6893.981,E2 -6893.981} C_VEL
LIN {X 0,Y 483.542,Z 667.088,A -85,B 0,C 180,E1 -6896.972,E2 -6896.972} C_VEL
LIN {X 0,Y 483.155,Z 679.461,A -85,B 0,C 180,E1 -6899.878,E2 -6899.878} C_VEL
LIN {X 0,Y 482.745,Z 694.056,A -85,B 0,C 180,E1 -6903.172,E2 -6903.172} C_VEL
LIN {X 0,Y 482.43,Z 706.601,A -85,B 0,C 180,E1 -6905.927,E2 -6905.927} C_VEL
LIN {X 0,Y 482.071,Z 721.819,A -85,B 0,C 180,E1 -6909.212,E2 -6909.212} C_VEL
LIN {X 0,Y 481.819,Z 736.871,A -85,B 0,C 180,E1 -6912.382,E2 -6912.382} C_VEL
LIN {X 0,Y 481.551,Z 749.381,A -85,B 0,C 180,E1 -6915.013,E2 -6915.013} C_VEL
LIN {X 0,Y 482.893,Z 762.392,A -85,B 0,C 180,E1 -6915.352,E2 -6915.352} C_VEL
LIN {X 0,Y 483.784,Z 770.014,A -85,B 0,C 180,E1 -6915.621,E2 -6915.621} C_VEL
